(* CODESYS project PPC-GD-14.xml

Project tree, tasks and I/O mapping:
  Alarm Configuration
    alarm class Alarm (priority 30, acknowledge REP)
    alarm class Critical (priority 0, acknowledge ACK)
    alarm class Warning (priority 50, acknowledge REP)
    alarm group InverterComms
    alarm group Measurement
    alarm group Protection
    alarm group Startup
        0 []: Comparison Equal
    alarm group StopTrip
    alarm group SystemWatchdog
    AlarmStorage
    text list InverterComms
    text list Measurement
    text list Protection
    text list Startup
    text list StopTrip
    text list SystemWatchdog
  DataTypes/
    data type E_EventCode
    data type E_FailState
    data type E_MachineState
    data type E_ModbusResult
    data type E_StartupStatus
    data type ST_Energia
    data type ST_EventEntry
    data type ST_Medidor
    data type ST_Rele
    data type TTraceEntry
    data type UN_Convert_Word_To_Real
    data type UN_Energia
    data type UN_Medidor
    data type UN_Real_to_Word_array
    data type UN_Rele
  Eventos/
    function block FB_EventLog [ST]: Clear, GetEvent, LogEvent
  FB Controle/
    function block FB_Controle [ST]
    function block FB_Diagnostico [ST]
    function block FB_DroopP [ST]
    function block FB_FFQ [ST]
    function block FB_FLimiter [ST]
    function block FB_PAlloc [ST]
    function block FB_PI [ST]
    function block FB_PIQ [ST]
    function block FB_PowerController [ST]
    function block FB_QAlloc [ST]
    function block FB_SafetyMargin [ST]
    function block FB_Scheduler [ST]
  FB Escrita/
    function block FB_WriteInv [ST]
  FB Leitura/
    function block FB_ReadMedidor [ST]
    function block FB_ValidaDadosMedidor [ST]
    function block FB_ValidaDadosRele [ST]
  Variaveis/
    global variables Global
    global variables GVL_Alarm
    global variables GVL_EventLog
    global variables GVL_Persis
  function block FB_Startup [ST]
  program MainProgram [ST]
  FB da IHM/
    function block FB_EventDisplay [ST]
    function FC_EpochToString [ST]
    function FC_EventCodeToString [ST]
    function FC_SeverityToString [ST]
    function FC_UIntToHex16Sharp [ST]
*)

// DataTypes/E_EventCode
{attribute 'qualified_only'}
{attribute 'strict'}
// ════════════════════════════════════════════════════════════════════
// E_EventCode — Código unificado de eventos do PPC-GD
// ════════════════════════════════════════════════════════════════════
//
// FAIXAS DE CÓDIGOS:
//   0x0000          = Sem evento
//   0x1xxx          = INFO     (informações operacionais)
//   0x2xxx          = WARNING  (desvios toleráveis, sem ação de potência)
//   0x4xxx          = ALARM    (falhas que requerem atenção ou degradam)
//   0x8xxx          = CRITICAL (ações de segurança: FAIL_SAFE ou STOP)
//
// SUB-FAIXAS (2º nibble = módulo):
//   x0xx = Sistema / Geral
//   x1xx = Startup (FB_Startup)
//   x2xx = Medição (FB_ReadMedidor, FB_ValidaDadosRele)
//   x3xx = Comunicação inversores (FB_WriteInv)
//   x4xx = Controle (FB_Controle, FB_PowerController, FB_PIQ)
//   x5xx = Scheduler / Agenda
//   x6xx = Máquina de Estados (MainProgram)
//   x7xx = Proteção normativa (timers 15s/30s, hard-limit)
//   x8xx = STOP / Trip
//   x9xx = Reservado para expansão
//   xAxx = Erros gerados pelo Driver Modbus do Codesys
//
// Observação: códigos legados (ex-16#C1/C2/E1/E2/E3/F1) são referenciados
// por comentário e mapeados semanticamente, sem manter o mesmo valor numérico,
// para preservar a coerência de severidade por faixa.
// ════════════════════════════════════════════════════════════════════
TYPE E_EventCode :
(
    EVT_NONE                        := 16#0000,

    // ══════════════════════════════════════════════════════════════
    // INFO (0x1xxx) — registro operacional, sem ação
    // ══════════════════════════════════════════════════════════════

    // ── Startup ──
    INFO_STARTUP_BEGIN              := 16#1100,  // Inicialização iniciada
    INFO_SERIAL_COM_OK              := 16#1101,  // COM1 e COM2 prontos
    INFO_RTC_OK                     := 16#1102,  // Relógio lido com sucesso
    INFO_INVERTER_COUNT             := 16#1103,  // Contagem de inversores concluída
    INFO_INSTALLED_POWER            := 16#1104,  // Potência instalada calculada
    INFO_K1_CONFIRMED               := 16#1105,  // K1_in confirmado (debounce)
    INFO_K2_CONFIRMED               := 16#1106,  // K2_in confirmado (debounce)
    INFO_STARTUP_DONE               := 16#1107,  // Startup completo → operação

    // ── Operação normal ──
    INFO_MEDIDOR_READ_OK            := 16#1200,  // Leitura do medidor OK
    INFO_MEDIDOR_DATA_VALID         := 16#1201,  // Dados validados e filtro aplicado
    INFO_MEAS_RECOVERING            := 16#1202,  // contador nErrors reduzindo (opcional)

    // ── Escrita inversores (0x13xx)
    INFO_WRITE_INV_OK               := 16#1300,  // Escrita em inversor OK

    // ── Scheduler (0x15xx)
    INFO_SPECIAL_DATE_ACTIVE        := 16#1500,  // Data especial ativa na agenda
    INFO_ZERO_GRID_MODE             := 16#1501,  // Modo Zero Grid ativo

    // ── Recuperação / Reset ──
    INFO_CYCLE_COMPLETE             := 16#1600,  // Ciclo READ→CONTROL→WRITE→IDLE OK
    INFO_FAIL_RECOVERY              := 16#1601,  // Recuperação automática do FAIL
    INFO_STATE_CHANGE               := 16#1610,  // Transição de MachineState

    // ── STOP/Reset (0x18xx)
    INFO_STOP_K2_OPEN_CONFIRMED     := 16#1800,  // K2 confirmado aberto no STOP
    INFO_STOP_RESET_APPROVED        := 16#1801,  // Reset manual aprovado
    INFO_STOP_RESET_WAITING         := 16#1802,  // Aguardando Pt estável para reset

    // ══════════════════════════════════════════════════════════════
    // WARNING (0x2xxx) — desvio tolerável, sem ação de potência
    // ══════════════════════════════════════════════════════════════

    // ── Startup ──
    WARN_TC_POWER_NOT_SET           := 16#2100,  // TC_Power_kW não configurado
    WARN_NO_INVERSORES_COM02        := 16#2101,  // COM2 sem inversores (pode ser intencional)

    // ── Medição ──
    WARN_MEAS_USING_LAST_VALID      := 16#2200,  // Usando última medição válida
    WARN_MEAS_CROSS_CHECK_PA        := 16#2201,  // Validação cruzada Pa inconsistente
    WARN_MEAS_CROSS_CHECK_PB        := 16#2202,  // Validação cruzada Pb inconsistente
    WARN_MEAS_CROSS_CHECK_PC        := 16#2203,  // Validação cruzada Pc inconsistente
    WARN_MEAS_CROSS_CHECK_PT_SUM    := 16#2204,  // Pt ≠ Pa+Pb+Pc
    WARN_MEAS_CROSS_CHECK_PF        := 16#2205,  // PFt inconsistente com P/S
    WARN_MEAS_ERROR_ISOLATED        := 16#2206,  // Erro de medição isolado (1-4 erros)

    // ── Comunicação inversores ──
    WARN_WRITE_INV_ERROR            := 16#2300,  // Erro escrita em inversor individual
    WARN_WRITE_INV_TIMEOUT          := 16#2301,  // Timeout escrita em inversor individual

    // ── Controle ──
    WARN_P_ALLOC_SATURATED          := 16#2400,  // P alocado < P comandado
    WARN_Q_LIMITED_BY_SMAX          := 16#2401,  // Q limitado por Smax dos inversores
    WARN_PF_BELOW_TARGET            := 16#2402,  // PF < 0.92 (mas não por limite de S)
    WARN_PF_NOT_ACHIEVABLE          := 16#2403,  // PF impossível (banco de capacitor)
    WARN_PI_P_SATURATED             := 16#2404,  // PI de P saturado
    WARN_PI_Q_SATURATED             := 16#2405,  // PI de Q saturado
    WARN_PHASE_LIMITED              := 16#2406,  // Potência limitada por fase

    // ── Ciclo ──
    WARN_SCAN_OVERRUN               := 16#2600,  // Ciclo excedeu tolerância (1x)

          // ── STOP/reset
    WARN_STOP_RESET_DENIED          := 16#2800,  // Reset manual negado

    // ══════════════════════════════════════════════════════════════
    // ALARM (0x4xxx) — falha que requer atenção, pode degradar
    // ══════════════════════════════════════════════════════════════

    // ── Medição — Range ──
    ALARM_MEAS_VOLTAGE_A_RANGE      := 16#4200,  // Tensão fase A fora de faixa
    ALARM_MEAS_VOLTAGE_B_RANGE      := 16#4201,  // Tens  o fase B fora de faixa
    ALARM_MEAS_VOLTAGE_C_RANGE      := 16#4202,  // Tensão fase C fora de faixa
    ALARM_MEAS_CURRENT_A_RANGE      := 16#4203,  // Corrente fase A fora de faixa
    ALARM_MEAS_CURRENT_B_RANGE      := 16#4204,  // Corrente fase B fora de faixa
    ALARM_MEAS_CURRENT_C_RANGE      := 16#4205,  // Corrente fase C fora de faixa
    ALARM_MEAS_PT_RANGE             := 16#4206,  // Potência total fora de faixa
    ALARM_MEAS_PA_RANGE             := 16#4207,  // Potência fase A fora de faixa
    ALARM_MEAS_PB_RANGE             := 16#4208,  // Potência fase B fora de faixa
    ALARM_MEAS_PC_RANGE             := 16#4209,  // Potência fase C fora de faixa
    ALARM_MEAS_QT_RANGE             := 16#420A,  // Reativa total fora de faixa
    ALARM_MEAS_QA_RANGE             := 16#420B,  // Reativa fase A fora de faixa
    ALARM_MEAS_QB_RANGE             := 16#420C,  // Reativa fase B fora de faixa
    ALARM_MEAS_QC_RANGE             := 16#420D,  // Reativa fase C fora de faixa
    ALARM_MEAS_PFT_RANGE            := 16#420E,  // PF total fora de faixa
    ALARM_MEAS_PFA_RANGE            := 16#420F,  // PF fase A fora de faixa
    ALARM_MEAS_PFB_RANGE            := 16#4210,  // PF fase B fora de faixa
    ALARM_MEAS_PFC_RANGE            := 16#4211,  // PF fase C fora de faixa
    ALARM_MEAS_FROZEN               := 16#4212,  // Medição congelada (Pt sem variação)

    // ── Comunicação medidor ──
    ALARM_MEDIDOR_MODBUS_ERROR      := 16#4220,  // Erro Modbus do medidor
    ALARM_MEDIDOR_TIMEOUT           := 16#4221,  // Timeout leitura medidor

    // ── Comunicação inversores ──
    ALARM_COM_CH1_DEGRADED          := 16#4300,  // Canal COM1 >50% falhas
    ALARM_COM_CH2_DEGRADED          := 16#4301,  // Canal COM2 >50% falhas
	
	// Erros gerados pelo Driver Modbus do Codesys
    ALARM_MB_ILLEGAL_FUNC         	:= 16#4A01,
    ALARM_MB_ILLEGAL_ADDR         	:= 16#4A02,
    ALARM_MB_ILLEGAL_VALUE        	:= 16#4A03,
    ALARM_MB_SLAVE_FAILURE        	:= 16#4A04,
    ALARM_MB_ACKNOWLEDGE          	:= 16#4A05,
    ALARM_MB_SLAVE_BUSY           	:= 16#4A06,
    ALARM_MB_MEMORY_PARITY        	:= 16#4A08,
    ALARM_MB_GW_PATH_UNAVAIL      	:= 16#4A0A,
    ALARM_MB_GW_DEVICE_FAIL       	:= 16#4A0B,
    ALARM_MB_RESPONSE_TIMEOUT     	:= 16#4AA1,
    ALARM_MB_RESPONSE_CRC         	:= 16#4AA2,
    ALARM_MB_WRONG_SLAVE          	:= 16#4AA3,
    ALARM_MB_WRONG_FC             	:= 16#4AA4,
    ALARM_MB_TCP_WARMOR           	:= 16#4AA5,
    ALARM_MB_INVALID_DATA         	:= 16#4AA6,
    ALARM_MB_INVALID_PROTOCOL     	:= 16#4AA7,
    ALARM_MB_INVALID_HEADER       	:= 16#4AA8,
    ALARM_MB_INVALID_PARAM        	:= 16#4AA9,
    ALARM_MB_UNDEFINED            	:= 16#4AFF,
	ALARM_MB_APP_ABORTED          	:= 16#4AB1,
    ALARM_MB_APP_TIMEOUT          	:= 16#4AB2,

    // ══════════════════════════════════════════════════════════════
    // CRITICAL (0x8xxx) — ação de segurança (FAIL_SAFE ou STOP)
    // ══════════════════════════════════════════════════════════════

    // ── Startup ──
    CRIT_SERIAL_INIT_FAILED         := 16#8100,  // COM1/COM2 não inicializou
    CRIT_RTC_FAILED                 := 16#8101,  // Falha leitura RTC
    CRIT_NO_INSTALLED_POWER         := 16#8102,  // Potência instalada = 0
    CRIT_K1_TIMEOUT                 := 16#8103,  // K1 não respondeu (timeout)

    // ── Medição ──
    CRIT_MEAS_PERSISTENT_FAIL       := 16#8200,  // ex-16#C1 Medição com falha persistente (≥5 erros)
    CRIT_MEDIDOR_COM_FAIL           := 16#8201,  // ex-16#C2 Erro/Timeout Modbus medidor → FAIL

    // ── Comunicação inversores ──
    CRIT_COM_CHANNEL_FAIL           := 16#8300,  // ex-16#C2 Canal COM com falha total → FAIL

    // ── Controle ──
    CRIT_INSTALLED_POWER_ZERO       := 16#8400,  // InstalledPower = 0 em runtime → STOP

    // ── Scheduller ──
    CRIT_RTC_READ_FAIL              := 16#8500,  // RTC falhou durante operação
    CRIT_SCHEDULE_INDEX_INVALID     := 16#8501,  // Índice dia/hora inválido

    // ── Watchdog ──
    CRIT_SCAN_WATCHDOG              := 16#8600,  // ex-16#F1 3× overruns consecutivos → FAIL

    // ── Proteção normativa ──
    CRIT_HARD_LIMIT_15S             := 16#8700,  // ex-16#E1 P > LPI+10%Pnom por >15s → STOP
    CRIT_EXPORT_OVER_LPI_30S        := 16#8701,  // ex-16#E2 P > LPI por >30s → STOP
    CRIT_MEDIDOR_TIMEOUT_IN_FAIL    := 16#8702,  // ex-16#E3 30s sem medição válida em FAIL → STOP

    // ── STOP / Trip ──
    CRIT_STOP_ENTRY                 := 16#8800,  // Entrada no estado STOP
    CRIT_K2_DID_NOT_OPEN            := 16#8801,  // K2 não abriu após 2s → FaultLatch
    CRIT_STATE_CORRUPTION           := 16#8802   // MachineState inválido

) UINT;
END_TYPE

// DataTypes/E_FailState
{attribute 'qualified_only'}
{attribute 'strict'}
TYPE E_FailState :
(
    FS_INIT         := 0,  // Inicialização FAIL_SAFE
    FS_FORCE_ZERO   := 1,  // Forçar setpoint zero
    FS_WAIT_CONFIRM := 2,  // Aguardar confirmação escrita
    FS_VALIDATE     := 3,  // Validar geração zero
    FS_ESCALATE     := 4   // Escalar para STOP
) UINT;
END_TYPE

// DataTypes/E_MachineState
{attribute 'qualified_only'}
{attribute 'strict'}
TYPE E_MachineState :
(
	START       := 0,  // inicializa o sistema uma única vez
    IDLE        := 1,  // Aguardando condições de início
    READ        := 2,  // Lendo medidor
    CONTROL     := 3,  // Calculando setpoints
    WRITE       := 4,  // Enviando comandos inversores
    FAIL	    := 5,  // Redução forçada (sem trip)
    STOP        := 6,   // Trip + latch (reset manual)
	ERROR       := 255 // Estado inválido/corrupto (fallback)
) UINT;
END_TYPE

// DataTypes/E_ModbusResult
{attribute 'strict'}
TYPE E_ModbusResult :
(
    BUSY,   	// operação em andamento
    DONE,   	// leitura finalizada com sucesso (pulso curto)
    ERRO,   	// falha (permanece até reset)
	ABORT,		// comunicação foi abortada
	TIMEOUT,	// ocorreu TIMEOUT
	END			// finaliza a comunicação
);
END_TYPE

// DataTypes/E_StartupStatus
{attribute 'qualified_only'}
{attribute 'strict'}
TYPE E_StartupStatus :
(
  stSeriais,		(* inicializa serias COM1 e COM2 *)
  stInit,			(* inicializa variaveis *)
  stWait_K1,      	(* transição imediata quando o delay completa *)
  stWait_K2,       	(* mantém bK3_out; monitora bK2_in com debounce *)
  stDone,           (* sucesso: desliga bK3_out e liga bK4_out *)
  stError           (* erro: sinaliza e coloca saídas em estado seguro *)
);
END_TYPE

// DataTypes/ST_Energia
TYPE ST_Energia :
	STRUCT
		// variavel       tipo      modbusAddress origem         fator_escala 
		EAImp  : REAL := 0.0; // 101EH - energia ativa total positiva (kWh)
		Vazia1 : REAL := 0.0; // 1020H - void
		Vazia2 : REAL := 0.0; // 1022H - void
		Vazia3 : REAL := 0.0; // 1024H - void
		Vazia4 : REAL := 0.0; // 1026H - void
		EAExp  : REAL := 0.0; // 1028H - energia ativa total negativa (kWh)	
	END_STRUCT
END_TYPE

// DataTypes/ST_EventEntry
// ════════════════════════════════════════════════════════════════════
// ST_Event — Registro individual de evento no ring buffer
// ════════════════════════════════════════════════════════════════════
// Tamanho estimado: 28 bytes (verificar alinhamento no target)
//
// CAMPOS:
//   tTimestamp  — Epoch UTC (UDINT, até 2106). Obtido via SysTimeRtcGet.
//   eCode      — Código do evento (E_EventCode). Identifica unicamente o que ocorreu.
//   bRaised    — TRUE = evento apareceu / FALSE = evento foi limpo.
//                Permite rastrear par raise/clear no histórico.
//   rParam1    — Valor de contexto #1 no momento do evento.
//                Ex: Pt medido (kW) quando hard-limit disparou.
//   rParam2    — Valor de contexto #2 no momento do evento.
//                Ex: limite violado (kW), ou índice do inversor.
//   uMachState — Estado da máquina (E_MachineState) no momento do registro.
//                Essencial para análise pós-mortem.
// ════════════════════════════════════════════════════════════════════
TYPE ST_EventEntry :
STRUCT
    tTimestamp      : UDINT;            // UTC epoch (segundos)
    eCode           : E_EventCode;      // UINT — código unificado do evento
    bRaised         : BOOL;             // TRUE=raise, FALSE=clear
    rParam1         : REAL;             // contexto numérico #1
    rParam2         : REAL;             // contexto numérico #2
    uMachState      : UINT;             // E_MachineState no instante do registro
END_STRUCT
END_TYPE

// DataTypes/ST_Medidor
TYPE ST_Medidor :
	STRUCT
		//  22 variaveis do tipo real - ocupam 44 Words no array
		// variavel       tipo      modbusAddress origem         fator_escala 
		Ua    	    : REAL := 0.0; // 2006H - Tensão de fase A x 0,1 V
		Ub    	    : REAL := 0.0; // 2008H - Tensão de fase B x 0,1 V
		Uc    	    : REAL := 0.0; // 200AH - Tensão de fase C x 0,1 V
		Ia    	    : REAL := 0.0; // 200CH - Corrente de fase A x 0,001 A 
		Ib    	    : REAL := 0.0; // 200EH - Corrente de fase B x 0,001 A
		Ic    	    : REAL := 0.0; // 2010H - Corrente de fase C x 0,001 A
		Pt    	    : REAL := 0.0; // 2012H - Potencia ativa combinada x 0,1 W
		Pa    	    : REAL := 0.0; // 2014H - Potencia ativa fase A x 0,1 W
		Pb    	    : REAL := 0.0; // 2016H - Potencia ativa fase B x 0,1 W
		Pc    	    : REAL := 0.0; // 2018H - Potencia ativa fase C x 0,1 W	
		Qt    	    : REAL := 0.0; // 201AH - Potencia reativa combinada x 0,1 var
		Qa    	    : REAL := 0.0; // 201CH - Potencia reativa fase A x 0,1 var
		Qb    	    : REAL := 0.0; // 201EH - Potencia reativa fase B x 0,1 var
		Qc    	    : REAL := 0.0; // 2020H - Potencia reativa fase C x 0,1 var
		Reserved01  : REAL;        // 2022H - sem informação
		Reserved02  : REAL;        // 2024H - sem informação
		Reserved03  : REAL;        // 2026H - sem informação
		Reserved04  : REAL;        // 2028H - sem informação
		PFt    	    : REAL := 0.0; // 202AH - Fator de potência combinado (número positivo: indutivo, número negativo: capacitivo) (x  0,001)
		PFa    	    : REAL := 0.0; // 202CH - Fator de potência de fase A (número positivo: indutivo, número negativo: capacitivo)  (×0,001)
		PFb    	    : REAL := 0.0; // 202EH - Fator de potência de fase B (número positivo: indutivo, número negativo: capacitivo)  (×0,001)
		PFc    	    : REAL := 0.0; // 2030H - Fator de potência de fase C (número positivo: indutivo, número negativo: capacitivo)  (×0,001)
	END_STRUCT
END_TYPE

// DataTypes/ST_Rele
TYPE ST_Rele :
	STRUCT
		//  22 variaveis do tipo real - ocupam 44 Words no array
		// variavel       tipo      modbusAddress origem         fator_escala 
		Ua    	    : REAL := 0.0; // 2006H - Tensão de fase A x 0,1 V
		Ub    	    : REAL := 0.0; // 2008H - Tensão de fase B x 0,1 V
		Uc    	    : REAL := 0.0; // 200AH - Tensão de fase C x 0,1 V
		Ia    	    : REAL := 0.0; // 200CH - Corrente de fase A x 0,001 A 
		Ib    	    : REAL := 0.0; // 200EH - Corrente de fase B x 0,001 A
		Ic    	    : REAL := 0.0; // 2010H - Corrente de fase C x 0,001 A
		Pt    	    : REAL := 0.0; // 2012H - Potencia ativa combinada x 0,1 W
		Pa    	    : REAL := 0.0; // 2014H - Potencia ativa fase A x 0,1 W
		Pb    	    : REAL := 0.0; // 2016H - Potencia ativa fase B x 0,1 W
		Pc    	    : REAL := 0.0; // 2018H - Potencia ativa fase C x 0,1 W	
		Qt    	    : REAL := 0.0; // 201AH - Potencia reativa combinada x 0,1 var
		Qa    	    : REAL := 0.0; // 201CH - Potencia reativa fase A x 0,1 var
		Qb    	    : REAL := 0.0; // 201EH - Potencia reativa fase B x 0,1 var
		Qc    	    : REAL := 0.0; // 2020H - Potencia reativa fase C x 0,1 var
		Reserved01  : REAL;        // 2022H - sem informação
		Reserved02  : REAL;        // 2024H - sem informação
		Reserved03  : REAL;        // 2026H - sem informação
		Reserved04  : REAL;        // 2028H - sem informação
		PFt    	    : REAL := 0.0; // 202AH - Fator de potência combinado (número positivo: indutivo, número negativo: capacitivo) (x  0,001)
		PFa    	    : REAL := 0.0; // 202CH - Fator de potência de fase A (número positivo: indutivo, número negativo: capacitivo)  (×0,001)
		PFb    	    : REAL := 0.0; // 202EH - Fator de potência de fase B (número positivo: indutivo, número negativo: capacitivo)  (×0,001)
		PFc    	    : REAL := 0.0; // 2030H - Fator de potência de fase C (número positivo: indutivo, número negativo: capacitivo)  (×0,001)
	END_STRUCT
END_TYPE

// DataTypes/TTraceEntry
TYPE TTraceEntry :
STRUCT
        cyc         : UDINT;
        mode        : USINT;
        startEdge   : BOOL;
        xExecute    : BOOL;
        xAbort      : BOOL;
        xBusy       : BOOL;
        xDone       : BOOL;
        xError      : BOOL;
        xAborted    : BOOL;
        toQ         : BOOL;
        modbusErr   : UDINT;
        eResult     : E_ModbusResult;
    END_STRUCT
END_TYPE

// DataTypes/UN_Convert_Word_To_Real
TYPE UN_Convert_Word_To_Real :
	UNION
        Tw : ARRAY[0..1] OF WORD;
        Tr : REAL;
    END_UNION
END_TYPE

// DataTypes/UN_Energia
TYPE UN_Energia :
	UNION
        WordArray : ARRAY[0..11] OF WORD;
        EmReal    : ST_Energia;
    END_UNION
END_TYPE

// DataTypes/UN_Medidor
TYPE UN_Medidor :
	UNION
        WordArray : ARRAY[0..43] OF WORD;
        EmReal    : ST_Rele;
    END_UNION
END_TYPE

// DataTypes/UN_Real_to_Word_array
TYPE UN_Real_to_Word_array :
UNION
	RealArr  : ARRAY[1..15] OF REAL;   // 60 bytes
    WordArr  : ARRAY[1..30] OF WORD;   // 60 bytes
END_UNION
END_TYPE

// DataTypes/UN_Rele
TYPE UN_Rele :
	UNION
        WordArray : ARRAY[0..43] OF WORD;
        EmReal    : ST_Rele;
    END_UNION
END_TYPE

// Variaveis/Global
{attribute 'qualified_only'}
VAR_GLOBAL CONSTANT

    // Parâmetros do sistema
    SOFTVERSION          		: UINT := 21;   				// Versão da aplicação
	DATAAPLICATION				: DATE := DATE#2025-12-05;		// Data da aplicação
	NMAXINVERSORES				: UINT := 30;					// Capacidade máxima de inversores
	TIPOSINVERSORES				: UINT := 8;					// total de inversores diferentes que podem estar presentes
	NDATASESPECIAIS 			: UINT := 48; 					// Quantidade de datas especiais disponíveis ao todo (para 10 anos)
	TIMEZONEOFFSET				: DINT := -3; 			
    CYCLE_TIME_MS				: UDINT := 1000;  				// tempo de ciclo de controle
	CYCLE_TIME_TOLERANCE		: UDINT := 1100;  				// tolerancia de ultrapassagem para tempo de ciclo de controle de 10%

END_VAR

VAR_GLOBAL
	timestampUTC				: UDINT;
	Result 						: RTS_IEC_RESULT;
  	ControlCycle    			: REAL;            					// Tempo de ciclo de controle em SEGUNDOS (ex: 1.0 = 1 segundo)
	
	// Saidas digitais
  	K1_out  					: BOOL;   							// DI X5_1 - K1 - controle permissivo
	K2_out						: BOOL;								// DI X5_2 - K2 - controle trip
  	K3RedOut					: BOOL;								// DI X5_3 - nada pronto - acende vermelho
  	K4YellowOut  				: BOOL;   							// DI X5_4 - K2 aberto - acende amarelo
  	K5GreenOut  				: BOOL;   							// DI X5_5 - K2 fechou - acende verde
	K7OkOut  					: BOOL;   							// DI X5_7 - sinaliza ok
	K8ErroOut  					: BOOL;   							// DI X5_8 - sinaliza erro
		
	// Entredas digitais
	K1_in        				: BOOL;                				// DI X12_1 - contato auxliar de K1
  	K2_in        				: BOOL;                				// DI X12_2 - contato auxliar de K2

    //    Medições (REAL) - Tensões (V), Correntes (A), Potências Ativas (W), Potências Reativas (var), PF (adimensional, sinal: + indutivo, - capacitivo)
	
    Ua  			: REAL := 0.0; // Tensão de fase A   - 2006H - Tensão de fase A em Volts (x 0,1 V)
    Ub  			: REAL := 0.0; // Tensão de fase B   - 2008H - Tensão de fase B em Volts (x 0,1 V)
    Uc  			: REAL := 0.0; // Tensão de fase C   - 200AH - Tensão de fase C em Volts (x 0,1 V)
	
	Ia    			: REAL 	:= 0.0; // 200CH - Corrente de fase A em A (x 0,001 A) 
	Ib    			: REAL 	:= 0.0; // 200EH - Corrente de fase B em A (x 0,001 A) 
	Ic    			: REAL 	:= 0.0; // 2010H - Corrente de fase C em A (x 0,001 A) 
	
	Pt    			: REAL 	:= 0.0; // 2012H - Potencia ativa combinada em kW (x 0.1 para W, x 0.0001 para kW)
	Pa    			: REAL 	:= 0.0; // 2014H - Potencia ativa fase A 	em kW (x 0.1 para W, x 0.0001 para kW)
	Pb    			: REAL 	:= 0.0; // 2016H - Potencia ativa fase B 	em kW (x 0.1 para W, x 0.0001 para kW)
	Pc    			: REAL 	:= 0.0; // 2018H - Potencia ativa fase C    em kW (x 0.1 para W, x 0.0001 para kW)

	Qt    			: REAL 	:= 0.0; // 201AH - Potencia reativa combinada em kvar (x 0.1 para var, x 0.0001 para kvar)
	Qa    			: REAL 	:= 0.0; // 201CH - Potencia reativa fase A	 em kvar (x 0.1 para var, x 0.0001 para kvar)
	Qb    			: REAL 	:= 0.0; // 201EH - Potencia reativa fase B	 em kvar (x 0.1 para var, x 0.0001 para kvar)
	Qc    			: REAL 	:= 0.0; // 2020H - Potencia reativa fase C	 em kvar (x 0.1 para var, x 0.0001 para kvar)
	
	PFt    			: REAL 	:= 0.0; // 202AH - Fator de potência combinado (número positivo: indutivo, número negativo: capacitivo) (x0,001)
	PFa    			: REAL 	:= 0.0; // 202CH - Fator de potência de fase A (número positivo: indutivo, número negativo: capacitivo) (x0,001)
	PFb    			: REAL 	:= 0.0; // 202EH - Fator de potência de fase B (número positivo: indutivo, número negativo: capacitivo) (x0,001)
	PFc    			: REAL 	:= 0.0; // 2030H - Fator de potência de fase C (número positivo: indutivo, número negativo: capacitivo) (x0,001)	

    //   COMANDOS E TELEMETRIA - Saídas do Controle 
	
	// definição dos inversores dos dois canais de comunicação
	
	trigInvCOM100  	: ARRAY[1..15] OF BOOL;
    pInversores100 	: ARRAY [1..15] OF POINTER TO ModbusSlaveComPort; 				// array de pointers para Inversor01..Inversor15 (apenas ponteiros - não recria instâncias)
	trigMedidor100 	: BOOL;
	pMedidor100		: POINTER TO ModbusSlaveComPort;
	
	trigInvCOM200  	: ARRAY[1..15] OF BOOL;
	pInversores200 	: ARRAY [1..15] OF POINTER TO ModbusSlaveComPort; 				// array de pointers para Inversor01..Inversor15 (apenas ponteiros - não recria instâncias)
	trigMedidor200 	: BOOL;
	pMedidor200		: POINTER TO ModbusSlaveComPort;
	
	// Potencia Total instalada e potencia Aparente Total instalada
  	InstalledPower 	: REAL; 														// Soma da potência nominal de todos os inversores ativos
	Q_max_permitido : REAL := 0.0;    												// Q máximo permitido (kvar)
	InstalledSmax   : REAL; 														// NOVO: Potência Aparente Máxima Total (kVA)	
	
	// COMANDOS DE CONTROLE
	MaxExportLimit 	: REAL;              											// Limite de exportação do scheduler (kW)
	P_cmd_total_kW 	: REAL;              											// Comando total de P (kW)
	Q_cmd_total_kvar: REAL;            												// Comando total de Q (kvar)
	
    
    // Telemetria: Setpoint atual da agenda (antes das proteções)
    TotalPowerPercent : REAL;

    // Telemetria: Potência Reativa total desejada (kVA)
    TotalReactivePower : REAL;

    // Telemetria: Valores efetivos calculados para cada inversor
    P_inv_kW     	: ARRAY[1..NMAXINVERSORES] OF REAL; 							// valor de setpoint de potencia ativa em kW
	P_inv_Percent 	: ARRAY[1..NMAXINVERSORES] OF REAL; 							// valor de setpoint de potencia ativa em percentual do nominal
    Q_inv_kvar    	: ARRAY[1..NMAXINVERSORES] OF REAL; 							// valor de setpoint de potencia reativa em kVA
    PF_inv 			: ARRAY[1..NMAXINVERSORES] OF REAL; 							// valor do fator de potencia de cada inversor (deve ser 0,92 para todos)
	P_inv_limit 	: ARRAY[1..NMAXINVERSORES] OF REAL; 							// valor limite de potencia ativa com base na SMAX de cada um
	
	// Margem de segurança para compensar erro de TC perto de zero, o sistema tentará manter importação mínima garantido que não haja exportação
	SafetyMargin_pct: REAL :=0.03;
	TC_Power_kW		: REAL := 0.0; // deve ser configurado como 3% da potencia total sob controle pelo TC
	
	// ════════════════════════════════════════════════════════════════
	// DIAGNÓSTICO DE PF
	// ════════════════════════════════════════════════════════════════
	Q_available_max : REAL;             											// Q máximo disponível (kvar)
	PF_effective 	: REAL;                											// PF efetivo resultante
	PFErro 			: BOOL;                   										// TRUE = PF < 0.92 não atingível (banco de capacitores)
    
	// ════════════════════════════════════════════════════════════════
    // DIAGNÓSTICO DE FATOR DE POTÊNCIA
    // ════════════════════════════════════════════════════════════════
    
    // Status geral
    PF_target : REAL := 0.92;                   // PF alvo (mínimo aceitável)
    PF_measured : REAL;                         // PF medido no ponto de conexão
    PF_achieved : REAL;                         // PF efetivamente alcançado após compensação
    PF_OK : BOOL;                               // TRUE = PF ≥ 0.92
    
    // Potências
    P_generated_kW : REAL;                      // P total gerado pelos inversores
    P_allocated_kW : REAL;                      // P efetivamente alocado
    Q_measured_kvar : REAL;                     // Q medido no ponto de conexão (carga)
    Q_required_kvar : REAL;                     // Q necessário para atingir PF ≥ 0.92
    Q_commanded_kvar : REAL;                    // Q comandado pelo FB_PIQ
    Q_available_kvar : REAL;                    // Q que inversores conseguem fornecer
    Q_allocated_kvar : REAL;                    // Q efetivamente alocado
    Q_deficit_kvar : REAL;                      // Déficit de Q (se > 0, falta Q)
    
    // Capacidade dos inversores
    S_total_available_kVA : REAL;               // S total disponível (soma de todos inversores)
    S_total_used_kVA : REAL;                    // S total utilizado
    S_utilization_pct : REAL;                   // % de utilização de S
    Q_capacity_total_kvar : REAL;               // Capacidade total de Q dos inversores (atual)
    Q_utilization_pct : REAL;                   // % de utilização de Q
    
    // Diagnóstico e recomendações
    Q_deficit_percent : REAL;                   // Déficit de Q em % do necessário
    Capacitor_bank_size_kvar : REAL;            // Tamanho recomendado de banco de capacitores
    Capacitor_bank_recommended : BOOL;          // TRUE = Recomenda banco de capacitores
    PF_alarm_code : UINT;                       // Código de alarme (0=OK, 1=Aviso, 2=Crítico)
    PF_alarm_message : STRING(255);             // Mensagem descritiva do alarme
    
    // Histórico (opcional)
    PF_min_24h : REAL := 1.0;                   // PF mínimo nas últimas 24h
    PF_avg_24h : REAL := 1.0;                   // PF médio nas últimas 24h
    Q_deficit_max_24h : REAL;                   // Déficit máximo de Q nas últimas 24h
    PF_alarm_count_24h : UDINT;                 // Quantidade de alarmes nas últimas 24h
    
    // Inversores individuais (diagnóstico detalhado)
    Inv_S_utilization : ARRAY[1..NMAXINVERSORES] OF REAL;  // % S usado por inversor
    Inv_Q_available : ARRAY[1..NMAXINVERSORES] OF REAL;    // Q disponível por inversor (kvar)
    Inv_limited : ARRAY[1..NMAXINVERSORES] OF BOOL;        // TRUE = Inversor limitado por S	
END_VAR

// Variaveis/GVL_Alarm
{attribute 'qualified_only'}
VAR_GLOBAL
    // ─────────────────────────────────────────────────────────
    // ALARM MANAGER FLAGS (condições booleanas)
    // ─────────────────────────────────────────────────────────
    // Medição / Medidor
    ALM_MEAS_MEDIDOR_TIMEOUT       	: BOOL := FALSE;  // timeout de leitura (READ)
    ALM_MEDIDOR_MODBUS_ERRO        	: BOOL := FALSE;  // xError do medidor (READ)
    ALM_MEAS_PERSISTENT_FAIL		: BOOL := FALSE;  // bPoucosErros = FALSE
    ALM_MEAS_FROZEN	                : BOOL := FALSE;  // diagnosticCode = A900 (se aplicável)
    ALM_MEAS_USING_LAST_VALUEU		: BOOL := FALSE;  // bPoucosErros=TRUE e bDadosOK=FALSE
	ALM_MEAS_RANGE_ERROR    		: BOOL := FALSE;    // Warning: Valor fora de faixa
    ALM_MEAS_XCHECK_FAIL   			: BOOL := FALSE;    // Warning: Validação cruzada falhou

    // Comunicação inversores
    ALM_MODBUS_COM1_FAIL        	: BOOL := FALSE;  // >50% falhas COM1 no ciclo
    ALM_MODBUS_COM2_FAIL            : BOOL := FALSE;  // >50% falhas COM2 no ciclo
    ALM_COM_CHANNEL_FAIL           	: BOOL := FALSE;  // falha geral de comunicação → FAIL/STOP

    // Sistema
	ALM_SCAN_OVERRUN        		: BOOL := FALSE;    // Warning: Watchdog de ciclo
    ALM_RTC_FAIL            		: BOOL := FALSE;    // Error: Falha RTC
    ALM_NO_INVERTERS        		: BOOL := FALSE;    // Error: Nenhum inversor configurado
    ALM_INSTALLED_PWR_ZERO  		: BOOL := FALSE;    // Error: Potência instalada = 0
    ALM_TC_POWER_NOT_SET            : BOOL := FALSE;    // PerVar.TC_Power_kW = 0 na inicialização

    // Proteções normativas
    ALM_HARDLIMIT_15S       		: BOOL := FALSE;    // Error: P > LPI+10% por >15s
    ALM_EXPORT_30S          		: BOOL := FALSE;    // Error: P > LPI por >30s
    ALM_K2_NOT_OPENED       		: BOOL := FALSE;    // Error: K2 não abriu após trip
	
	// Status do sistema
    ALM_STOP_ACTIVE	                : BOOL := FALSE;  	// MachineState=STOP
	ALM_FAIL_ACTIVE					: BOOL := FALSE;  	// MachineState=FAIL

    // ── Controle / PF ──
    ALM_PF_BELOW_TARGET     		: BOOL := FALSE;    // Warning: PF < 0.92
    ALM_PF_CRITICAL         		: BOOL := FALSE;    // Error: PF < 0.92 + Q saturado
    ALM_Q_SATURATED         		: BOOL := FALSE;    // Info: Q limitado por S
END_VAR

// Variaveis/GVL_EventLog
{attribute 'qualified_only'}
// ════════════════════════════════════════════════════════════════════
// GVL_EventLog — Constantes do sistema de log de eventos
// ════════════════════════════════════════════════════════════════════
// Autor: Eng. Principal / Revisão Técnica PPC-GD
// Plataforma: WAGO CC100 (751-9402) / CODESYS V3.5 SP21 Patch 4
//
// DIMENSIONAMENTO:
//   64 entradas × 28 bytes = ~1.792 bytes de RETAIN
//   WAGO CC100 possui ~32 kB RETAIN → uso < 6%
//   Com ~1 evento/min, cobre >1 hora de histórico completo
//   Com taxa de pico (~10 eventos em cascata), ainda retém >6 min
// ════════════════════════════════════════════════════════════════════
{attribute 'qualified_only'}
VAR_GLOBAL CONSTANT
    MAX_EVENT_ENTRIES   : UINT := 64;   // Tamanho do ring buffer (potência de 2 facilita debug)
END_VAR

// Variaveis/GVL_Persis
{attribute 'qualified_only'}
VAR_GLOBAL PERSISTENT RETAIN

    // CONFIGURAÇÕES DO SISTEMA (Dados que não podem ser perdidos no desligamento)
    
    // --- Configuração dos Inversores ---
	NInversoresCOM01    : UINT :=0;
	NInversoresCOM02    : UINT :=0;
	
    // Potência nominal (kW) por tipo
    InvActivePower 		: ARRAY[1..Global.NMAXINVERSORES] OF REAL; 		// kW
    // Potência Aparente Máxima (kVA) por tipo 
    InvSmaxPower 		: ARRAY[1..Global.NMAXINVERSORES] OF REAL;		// kVA

    // --- Parâmetros de Controle de Exportação ---
    PowerMode 			: UINT := 2;      								// 0=Total, 1=Por Fase, 2=Ambos
	OperationMode		: BOOL := TRUE;									// FALSE=Export Control  TRUE=Zero Grid
	ControlMode			: UINT := 1;									// 0 = manual  1 = automatico (PI ativo)
    TotalMaxExport_kW 	: REAL := 0; 									// Limite físico total (kW)
    PhaseMaxExport_kW 	: REAL := 0; 									// Limite físico por fase (kW)

    (* 
	Regra prática para GD solar: Ti entre 5s e 20s. Mais rápido pode oscilar com a latência Modbus. 
	Mais lento perde capacidade de compensar nuvens passando.
	Ti é o Tempo Integral do controlador PI, também chamado de tempo de reset.
	Relação Ki= Kp / Ti   Então se você tem Kp = 1.0 e Ti = 10s => Ki=1.0/10 = 0.1 (por segundo)
	Na prática para seu sistema:
	Ti pequeno (ex: 2s) → integral age rápido → mais agressivo → risco de oscilação
	Ti grande (ex: 30s) → integral age devagar → mais conservador → lento para corrigir erro estacionário
	Ti = 10s → o controlador elimina o erro estacionário em aproximadamente 30 a 40 segundos (≈ 3-4 × Ti)
	Resumo em uma frase:
	Ti = 10s é "quanto tempo o integrador leva para alcançar a mesma força que o proporcional já deu instantaneamente".
	*)
	
	// --- Controle Droop (Potência Ativa) ---
	Droop_Enable     	: BOOL := TRUE;      							// Habilita droop
	K_Droop          	: REAL := 0.15;      							// kW/kW  (ex.: 0.05 = 5% de ganho)
	Deadband_Droop   	: REAL := 2.0;       							// % (erro menor não gera droop)
	Droop_Max        	: REAL := 0.4;       							// Fração da potência instalada (ex.: 0.6 = 60%)
	
	// --- Parâmetros do Controlador PI (Potência Ativa) ---
    Kp_P           		: REAL := 0.25;									// Recomendado: 0.1 a 1.0
																	    // Maior → resposta mais rápida, risco de oscilação
																	    // Menor → mais suave, mas mais lento
    Ki_P           		: REAL := 0.02;									// Recomendado: 0.02 a 0.1 - Com 1s de ciclo e tempo morto ~1,2–1,6s, integral muito alto oscila.
																		// Com T=1s: constante de tempo integral Ti = Kp/Ki = 12,5s
																	    // Significado: elimina erro estacionário em ~10 segundos
																	    // NUNCA > 0.2 com T=1s (oscilação garantida)
	RampUp_P 			: REAL := 15.0;           						// Rampa de subida (kW/s) - limitar a 15-20 kW/s por causa do sweep de setpoints nos inversores
	RampDown_P 			: REAL := 20.0;         						// Rampa de descida (kW/s) - RampDown_P ≤ 20–30 kW/s
    Deadband_P  		: REAL := 1.0;  								// % da potência instalada (ex: 1.0 = 1%)
	
    // --- Configuração de Fator de Potência (PF) e Reativos (Q) ---
    PF_target       	: REAL := 0.92; 								// Alvo |PF|
	PF_sign				: REAL := 1.0;
    // Parâmetros do PI de Correção de Q (Feedforward + Feedback)
    Kp_Q           		: REAL := 50.0;									// Recomendado: 20.0 a 100.0 kvar/pu_PF
																	    // Unidade: kvar por unidade de erro de PF
																	    // Ex: erro PF = 0.02 → P_term = 50 * 0.02 = 1.0 kvar
    Ki_Q           		: REAL := 5.0;									// Recomendado: 2.0 a 10.0 kvar/(pu_PF·s
																	    // Com T=1s: Ti = Kp/Ki = 10s => elimina erro em ~30-40s
																	    // Significado: corrige PF em ~10 segundos	
	RampUp_Q 			: REAL := 50.0;            						// Rampa de subida (kvar/s)
	RampDown_Q 			: REAL := 50.0;          						// Rampa de descida (kvar/s)
	Deadband_Q 			: REAL := 0.01;          						// Zona morta de PF (ex: 0.01 = ±0.01) — padrão para GD

    // --- Histerese de Habilitação ---
    HysteresisOn	   	: REAL := 0.01; 								// Liga controle acima de 1%
    HysteresisOff		: REAL := 0.01; 								// Desliga abaixo de 1%
		
    // --- Agenda Semanal (7 dias x 24 horas) e Datas Especiais
	bHorarioVerao 		: BOOL:= FALSE;									// se TRUE  = Horário de Verão Ativo (+1h)
    WeekSchedule_kW 	: ARRAY[1..7, 1..24] OF REAL; 					// (1=Dom 2=Seg 3=Ter 4=Quarta 5=Quinta 6=Sexta 7=Sábado) em kW
    DatasEspeciais   	: ARRAY[1..GLOBAL.NDATASESPECIAIS] OF DATE;		// inicializa com zeros
	SpecialDaySchedule 	: ARRAY[1..Global.NDATASESPECIAIS] OF REAL;		// cada data especial tem apenas um valor de potencia maxima valido para o dia inteiro

    // ════════════════════════════════════════════════════════════════
    // LIMITES FÍSICOS DO SISTEMA (Baseados no Transformador e Rede)
    // ════════════════════════════════════════════════════════════════
	// SafetyMargin_kW = SafetyMargin_pct × TC_Power_kW / 100 - Margem de segurança para compensar erro de TC perto de zero
	SafetyMargin_pct 	: REAL := 3.0;     								// Percentual do TC (%)
	// Exemplo 1: TC de 500 A, Tensão 380 V => P_TC = √3 × V × I = 1.732 × 380 × 500 = 329 kW
	TC_Power_kW			: REAL := 0.0; 									// deve ser configurado como 3% da potencia total sob controle pelo TC
	
	VMIN 				: REAL := 7170;  // Volts - tensão de fase minima para tensão primária de 13,8kV
    VMAX 				: REAL := 8370;  // Volts - tensão de fase máxima para tensão primária de 13,8kV
    IMAX 				: REAL := 125.0;  // Amperes - corrente de linha - para potencia de usina de 3MW erro transformador 5%
    PMAX 				: REAL := 3200.0; // kW (Demanda contratada + 10% de margem)
	QMAX				: REAL := 2400.0; // kvar tan(acos(0.8)) × Pmax
	// τ = tempo para atingir ~63% do valor final e T_scan = período de amostragem (1s no seu caso)
	// α = T_scan / (τ + T_scan)  => Alpha=0.5 => 3 segundos para atingir 95% do valor final
	// Item 2.1: "Responder em até 15 segundos a rejeição de carga"
	// Item 2.2: "Limitar exportação em até 15 segundos"
	// Nuvens passageiras: variação em 1–5 segundos
	// Rejeição de carga: instantânea (< 1s)
	// Ruído de medição: < 100 ms
	ALPHA				: REAL := 0.25;
	
END_VAR

// FB_Startup
(* FB: fbStartup
   1) Ativa K1_out
   2) Aguarda 400 ms antes de verificar se K1_in está ativo
      -> Se K1_in NÃO estiver ativo depois deste tempo, sinaliza erro e sai da fbStartup
   3) Monitorar K2_in com debounce até ficar ativo 
   4) Enquanto aguarda K2_in ativar, mantém K4_out ativo
   5) Quando K2_in ativar (após debounced), desativa K4_out e ativa K5_out
   6) O controlador aguarda até K2_in = TRUE
   Notas:
   	- IMPORTANTE: se não forem usados contados auxiliares nos disjuntores, K1_in e K2_in precisam ser conectados a 24V
	- Este FB apenas sinaliza os outputs K1_out, K3_out, K4_out e K5_out.
   	- Implementado com máquina de estados e TONs (tDelay e tDebounce). TON deve ser chamado toda iteração.  *)
   
FUNCTION_BLOCK FB_Startup
VAR_OUTPUT
  stState			: E_StartupStatus:= E_StartupStatus.stSeriais;
END_VAR

VAR
  fbChannel       	: ModbusChannel;
  debouncedK1     	: BOOL := FALSE;   								// flag auxiliar informando que K1_in está estável em 1 
  TonDebounceK1     : TON;                          				// Novo timer debounce K1_in
  TimeDebounceK1    : TIME := T#500MS;              				// Tempo de debounce para K1

  debouncedK2 		: BOOL := FALSE; 								// flag auxiliar informando que K2_in está estável em 1 
  TonDebounceK2 	: TON;   										// timer para debounce de bk2 
  TimeDebounceK2    : TIME := T#500MS;     							// tempo de debounce para leitura de K2_in 
  
  cmdK01     		: BOOL := FALSE;  								// comandos calculados por ciclo e aplicados no final 
  auxRed     		: BOOL := FALSE;
  auxYellow     	: BOOL := FALSE;
  auxGreen     		: BOOL := FALSE;
  auxK1_in  		: BOOL;											// entradas digitais lidas no inicio da função 
  auxK2_in			: BOOL;
  indice			: UINT;
  
  // Variáveis para o Master 01 (COM1)
  eDeviceState01     		: DED.DEVICE_STATE; 					// Para guardar o estado retornado
  xDiagInfoIsAvailable01 	: BOOL;            						// Para guardar a saída xDiagnosisInfoAvailable
  eError01	      	    	: DED.ERROR;        					// Para guardar o código de erro
  xMaster01IsReady   		: BOOL;            						// Nosso booleano final de "pronto"
  
  // Variáveis para o Master 02 (COM2)
  eDeviceState02     		: DED.DEVICE_STATE; 					// Para guardar o estado retornado
  xDiagInfoIsAvailable02 	: BOOL;            						// Para guardar a saída xDiagnosisInfoAvailable
  eError02	           		: DED.ERROR;        					// Para guardar o código de erro
  xMaster02IsReady   		: BOOL;            						// Nosso booleano final de "pronto"
 

END_VAR

// INICIA AQUI

auxK1_in := Global.K1_in;
auxK2_in := Global.K2_in;

TonDebounceK1(IN := (stState = E_StartupStatus.stWait_K1) AND auxK1_in, PT := TimeDebounceK1); 	// debounce para K1_in
TonDebounceK2(IN := (stState = E_StartupStatus.stWait_K2) AND auxK2_in, PT := TimeDebounceK2);  // debounce para K2_in

CASE stState OF 																				// Máquina de estados

	E_StartupStatus.stSeriais:
		eDeviceState01 := Master_01.GetDeviceState(
			xDiagnosisInfoAvailable => xDiagInfoIsAvailable01,
			eError                  => eError01
			);
		eDeviceState02 := Master_02.GetDeviceState(
			xDiagnosisInfoAvailable => xDiagInfoIsAvailable02,
			eError                  => eError02
			);
  		xMaster01IsReady := (eDeviceState01 = DED.DEVICE_STATE.RUNNING); 
   		xMaster02IsReady := (eDeviceState02 = DED.DEVICE_STATE.RUNNING); 
		
		IF xMaster01IsReady AND xMaster02IsReady THEN
			stState := E_StartupStatus.stInit;
		ELSE
			stState := E_StartupStatus.stSeriais;
			// dispara Alarme por não conseguir abrir seriais
		END_IF
		
  	E_StartupStatus.stInit:																		// Inicialização única
	   
		cmdK01 			:= FALSE;
		auxRed  		:= FALSE;
		auxYellow 		:= FALSE;
		auxGreen  		:= FALSE;
		debouncedK1 	:= FALSE;
		debouncedK2 	:= FALSE;
		
		// Testa leitura do relógio do sistema na inicialização
		Global.timestampUTC := TO_UDINT(SysTimeRtcGet(Global.Result)); 							// UDINT#1528268918
		IF Global.Result <> eResultCode.OK THEN 												// Em caso de erro de leitura do relógio, zera a saída por segurança
			// sinalizar que houve erro para ler o relógio
			Global.K8ErroOut:=TRUE;
			RETURN;
		END_IF
	
		// Porta de comunicação COM1
		Global.pMedidor100   		:= ADR(Medidor100);
		Global.pInversores100[1]  	:= ADR(Inversor101);
		Global.pInversores100[2]  	:= ADR(Inversor102);
		Global.pInversores100[3]	:= ADR(Inversor103);
		Global.pInversores100[4] 	:= ADR(Inversor104);
		Global.pInversores100[5]	:= ADR(Inversor105);
		Global.pInversores100[6] 	:= ADR(Inversor106);
		Global.pInversores100[7] 	:= ADR(Inversor107);
		Global.pInversores100[8] 	:= ADR(Inversor108);
		Global.pInversores100[9] 	:= ADR(Inversor109);
		Global.pInversores100[10]	:= ADR(Inversor110);
		Global.pInversores100[11]	:= ADR(Inversor111);
		Global.pInversores100[12] 	:= ADR(Inversor112);
		Global.pInversores100[13] 	:= ADR(Inversor113);
		Global.pInversores100[14] 	:= ADR(Inversor114);
		Global.pInversores100[15] 	:= ADR(Inversor115);
		
		// Porta de comunicação COM2
		Global.pMedidor200   	  	:= ADR(Medidor200);
		Global.pInversores200[1]  	:= ADR(Inversor201);
		Global.pInversores200[2]  	:= ADR(Inversor202);
		Global.pInversores200[3]  	:= ADR(Inversor203);
		Global.pInversores200[4]  	:= ADR(Inversor204);
		Global.pInversores200[5] 	:= ADR(Inversor205);
		Global.pInversores200[6]  	:= ADR(Inversor206);
		Global.pInversores200[7]  	:= ADR(Inversor207);
		Global.pInversores200[8]  	:= ADR(Inversor208);
		Global.pInversores200[9]  	:= ADR(Inversor209);
		Global.pInversores200[10] 	:= ADR(Inversor210);
		Global.pInversores200[11] 	:= ADR(Inversor211);
		Global.pInversores200[12] 	:= ADR(Inversor212);
		Global.pInversores200[13] 	:= ADR(Inversor213);
		Global.pInversores200[14] 	:= ADR(Inversor214);
		Global.pInversores200[15] 	:= ADR(Inversor215);
		
		FOR indice := 1 TO 15 DO														// inicialização dos canais de comunicação
			fbChannel(Slave := Global.pInversores100[indice]^,xExecute := FALSE,xAbort := FALSE,iChannelIndex := 0);
			fbChannel(Slave := Global.pInversores200[indice]^,xExecute := FALSE,xAbort := FALSE,iChannelIndex := 0); 
		END_FOR
	
		// =========================================================================================
		// 0. PREPARAÇÃO DO TEMPO DE CICLO - feito na inicialização
		// =========================================================================================
		// Converte TIME (ex: T#500ms) para REAL (0.5 segundos) para uso nos PIDs
		Global.ControlCycle := UDINT_TO_REAL(Global.CYCLE_TIME_MS)/1000;  				// converte para segundos
			
		// ============================================================
		// CONTAGEM AUTOMÁTICA DE INVERSORES (sequencial por potência)
		// ============================================================
		
		// COM1: índices 1..15
		GVL_Persis.NInversoresCOM01 := 0;
		FOR indice := 1 TO 15 DO
			IF GVL_Persis.InvActivePower[indice] > 0.0 THEN
				GVL_Persis.NInversoresCOM01 := indice;   // mantém maior índice válido
			ELSE
				EXIT;  // encontrou buraco -> encerra contagem
			END_IF
		END_FOR
		
		// COM2: índices 16..30
		GVL_Persis.NInversoresCOM02 := 0;
		FOR indice := 16 TO 30 DO
			IF GVL_Persis.InvActivePower[indice] > 0.0 THEN
				GVL_Persis.NInversoresCOM02 := indice - 15;   // converte para faixa 1..15
			ELSE
				EXIT;  // encontrou buraco -> encerra contagem
			END_IF
		END_FOR		
		
		// =========================================================================================
		// 1. CÁLCULO DA POTÊNCIA INSTALADA TOTAL (Ativa e Aparente)  - feito na inicialização
		// =========================================================================================
		// Soma a capacidade nominal de todos os inversores configurados.
		// Isso permite mudar a planta dinamicamente sem recompilar.
		
		Global.InstalledPower := 0.0;
		Global.InstalledSmax  := 0.0;
		
		FOR indice := 1 TO Global.NMAXINVERSORES DO
			// Soma Potência Ativa Máxima (kW)
			Global.InstalledPower := Global.InstalledPower + GVL_Persis.InvActivePower[indice];
			// Soma Potência Aparente Máxima (kVA)
			Global.InstalledSmax := Global.InstalledSmax + GVL_Persis.InvSmaxPower[indice];
		END_FOR

		// Se não houver inversores ou potência válida, zera tudo e sai.
		IF Global.InstalledPower <= 0.0 THEN
			Global.TotalReactivePower := 0.0;
			// SINALIZA ALARME
			Global.K8ErroOut:=TRUE;
			RETURN;
		END_IF
		
		// Calcula Q_max_permitido 
	    Global.Q_max_permitido := Global.InstalledPower * 0.4256;  // tan(acos(0.92))
			
		// Configura TC_Power_kW se não foi configurado
		IF GVL_Persis.TC_Power_kW = 0.0 THEN
			// SINALIZA ALARME
			Global.K8ErroOut:=TRUE;
			GVL_Persis.TC_Power_kW := Global.InstalledPower;  // Aproximação conservadora
		END_IF

		// Muda para próximo estado	
		stState := E_StartupStatus.stWait_K1;

  E_StartupStatus.stWait_K1:															// DEBOUNCE K1
  
		cmdK01 := TRUE;
		auxRed := TRUE;																	// Status: aguardando K1 com debounce
		auxYellow := FALSE;
		auxGreen := FALSE;
		IF TonDebounceK1.Q THEN
		  debouncedK1 := TRUE;
		ELSE
		  debouncedK1 := FALSE;
		END_IF
	
		IF debouncedK1 THEN
		  stState := E_StartupStatus.stWait_K2;												// Somente avança se K1 está estabilizado
		  debouncedK2 := FALSE;
		  TonDebounceK1(IN := FALSE, PT := TimeDebounceK1); 								// (Opcional) reseta timer
		  auxRed := FALSE;																	// Status: aguardando K1 com debounce
		  auxYellow := TRUE;
		  auxGreen := FALSE;
		  
		END_IF

  E_StartupStatus.stWait_K2:	
  
		IF TonDebounceK2.Q THEN																// tDebounce.Q será TRUE se K2_in estável
		  debouncedK2 := TRUE;
		ELSE     																					
		  debouncedK2 := FALSE;																// se K2_in voltar a false, reseta timer
		END_IF
	
		IF debouncedK2 THEN
		  stState := E_StartupStatus.stDone;												// K2_ok e estável, processo de startup completo
		  TonDebounceK2(IN := FALSE, PT := TimeDebounceK2); 								// (Opcional) reseta timer
		  auxRed := FALSE;																	// Status: aguardando K1 com debounce
		  auxYellow := FALSE;
		  auxGreen := TRUE;
		END_IF
	
	E_StartupStatus.stDone:
	
		stState := E_StartupStatus.stDone;
		auxRed := FALSE;		
		auxYellow := FALSE;
		auxGreen := TRUE;

END_CASE;

//   Aplicar comandos calculados às saídas físicas / públicas
Global.K1_out 		:= cmdK01;
Global.K3RedOut 	:= auxRed;
Global.K4YellowOut 	:= auxYellow;
Global.K5GreenOut 	:= auxGreen;

END_FUNCTION_BLOCK

// MainProgram
// DEBUG
// {#define DEBUG_MODE}
PROGRAM MainProgram
(*
    Máquina de estados principal do controlador.
    Fluxo geral:
    START   -> READ    (quando fbStart termina com sucesso)
    READ    -> CONTROL (quando leitura Modbus do medidor conclui OK)
    READ    -> IDLE    (quando leitura falha, mas ainda não estourou RETRIES_READ)
    READ    -> FAIL    (quando leitura falha e estoura RETRIES_READ)
    CONTROL -> WRITE   (sempre, um ciclo de controle por leitura)
    WRITE   -> IDLE    (depois de tentar escrever em todos inversores, se não estourou RETRIES_WRITE)
    WRITE   -> FAIL    (se falhas de escrita estourarem RETRIES_WRITE)
    IDLE    -> READ    (quando completar 1 segundo de ciclo)
    FAIL    -> (aguarda ação do operador)
    STOP    -> (parada controlada, permanece travado)
*)

VAR
    fbStart         		: FB_Startup;        		// executa a inicialização
    fbControle      		: FB_Controle;		 		// módulo de controle
	fbAlarmes				: FB_Alarmes;		 		// converte códigos de erros em mensagens texto
	fbChannel       		: ModbusChannel;
	fbReadMedidor 			: FB_ReadMedidor;
	fbWriteInvCOM1 			: FB_WriteInv;
    fbWriteInvCOM2 			: FB_WriteInv;
	fbEventLog 				: FB_EventLog;    			// Instância única do ring buffer
    fbEventDisplay  		: FB_EventDisplay;			// prepara dados para a IHM
	
	// ══════════════════════════════════════════════════════════
    // Máquina de Estados
    // ══════════════════════════════════════════════════════════
	MachineState 			: E_MachineState := E_MachineState.START;
	MachineState_Last 		: E_MachineState := E_MachineState.START;
    FailState     			: E_FailState := E_FailState.FS_INIT;
	
	// ══════════════════════════════════════════════════════════
	// Variáveis manipuladas pela IHM
	// ══════════════════════════════════════════════════════════
 	HMI_bRefresh    : BOOL;     // Botão "Refresh" na IHM (pulso)
    HMI_nPage       : UINT;     // Página atual (0 = mais recente)
	
    // ══════════════════════════════════════════════════════════
    // STOP: Trip e Reset Manual
    // ══════════════════════════════════════════════════════════
    StopLatch         : BOOL := FALSE;
    StopResetCmd      : BOOL := FALSE;
    StopEntryTime     : UDINT := 0;
    K2_CheckDone      : BOOL := FALSE;
    sMessage_K2       : STRING(100) := '';
    bResetConditionsOK: BOOL := FALSE;
    sResetDenialReason: STRING(255) := '';
    rTrigReset        : R_TRIG;
    tonResetWindow    : TON;
    
    // ══════════════════════════════════════════════════════════
    // Timers Normativos (DIS-NOR-033)
    // ══════════════════════════════════════════════════════════
    ton15s  : TON;   // Hard limit > 15s → STOP
    ton30s  : TON;   // Exportação > LPI por > 30s → STOP
    ton2s   : TON;   // Confirmação K2 aberto

    // ══════════════════════════════════════════════════════════
    // Health Monitoring
    // ══════════════════════════════════════════════════════════
    MedidorOK         : BOOL := FALSE;
    ComOK             : BOOL := FALSE;
    ComOK_COM1        : BOOL := TRUE;
    ComOK_COM2        : BOOL := TRUE;
    InvOnlineCount    : UINT := 0;
    ScanOverrunCount  : UINT := 0;
	FaultLatch        : BOOL := FALSE;
	
    // ══════════════════════════════════════════════════════════
    // Limites Calculados
    // ══════════════════════════════════════════════════════════
    LPI_per_phase_kW  : REAL := 0.0;
    HardLimit_mag     : REAL := 0.0;
    LPI_mag			  : REAL;
	Export_mag		  : REAL;
    // ══════════════════════════════════════════════════════════
    // Validação Cruzada
    // ══════════════════════════════════════════════════════════
    Pt_Last           : REAL := 0.0;
    P_inv_sum         : REAL := 0.0;
    
    // ══════════════════════════════════════════════════════════
    // Escrita em Inversores (Sequencial)
    // ══════════════════════════════════════════════════════════
    InvIndexCOM1      : UINT := 1;
    InvIndexCOM2      : UINT := 1;
    ErrorCountCOM1    : UINT := 0;
    ErrorCountCOM2    : UINT := 0;
    DoneCOM1          : BOOL := FALSE;
    DoneCOM2          : BOOL := FALSE;
    LastErrorIdxCOM1  : UINT := 0;
    LastErrorIdxCOM2  : UINT := 0;
    WriteErrorCOM1    : BOOL := FALSE;
    WriteErrorCOM2    : BOOL := FALSE;
    
    // ══════════════════════════════════════════════════════════
    // Temporização e Watchdog
    // ══════════════════════════════════════════════════════════
    tCycleStart       : UDINT := 0;
    tCycleEnd         : UDINT;
    tCycle            : UDINT;
    tElapsed          : UDINT;
    bFirstScanRead    : BOOL := TRUE;
    MaxCycleTime      : UDINT := 0;
    CycleTimeOverrunCount : UDINT := 0;
    
    // ══════════════════════════════════════════════════════════
    // Debug/Monitor
    // ══════════════════════════════════════════════════════════
    valor             : UN_Convert_Word_To_Real;
    auxvalor          : REAL := 0;
    stStart, stEnd, stCiclo : SYSTIME;
    tStartCom, tCom, tEndCom: SYSTIME;
    tMax              : SYSTIME := 0;
    Gatilho           : BOOL := TRUE;
    rTrigOn           : R_TRIG;
    fTrigOff          : F_TRIG;
    Primeiravez       : BOOL := TRUE;
    stCicloMax        : SYSTIME := 0;
    i                 : UINT;
    
    // ══════════════════════════════════════════════════════════
    // FAIL_SAFE (STOP Timeout)
    // ══════════════════════════════════════════════════════════
    tonStopWrite      : TON;
    tStopWrite        : TIME := T#2S;


	tonFailSafeRecovery		: TON;   // tempo para recuperação ao normal
	tonMedidorTimeout		: TON;   // tempo que aguarda medidor sem leitura
    
END_VAR

// Chama o FB de display todo ciclo (ele só recalcula quando HMI_bRefresh der pulso)
fbEventDisplay(
    pEventLog   := fbEventLog,     // referência ao ring buffer
    bRefresh    := HMI_bRefresh,   // pulso da IHM
    nPageOffset := HMI_nPage       // página selecionada
);


// ════════════════════════════════════════════════════════════════
// MÁQUINA DE ESTADOS PRINCIPAL
// ════════════════════════════════════════════════════════════════
CASE MachineState OF
	
// ────────────────────────────────────────────────────────────────
// START: Inicialização (fbStart + K1/K2)
E_MachineState.START:
    fbStart();  // Chamada do bloco de inicialização
	
	CASE fbStart.stState OF
  		E_StartupStatus.stSeriais,
		E_StartupStatus.stInit,
        E_StartupStatus.stWait_K1,
        E_StartupStatus.stWait_K2:
        	// Permanece em START
        E_StartupStatus.stDone:
			// Inicialização única (executada 1x após power-on)
			FailState := E_FailState.FS_INIT;
			FaultCode := 0;
			FaultLatch := FALSE;
			StopLatch := FALSE;
			ton15s(IN := FALSE);
			ton30s(IN := FALSE);
			ton2s(IN := FALSE);
            (* Inicialização concluída – segue para leitura *)		
            MachineState := E_MachineState.READ;

{#ifdef DEBUG_MODE}			
MachineState := E_MachineState.CONTROL;
auxvalor:=0;
{#endif}
	END_CASE;

// ────────────────────────────────────────────────────────────────
// READ: Leitura do Medidor
E_MachineState.READ:

    // Marca início do ciclo apenas uma vez ao entrar em READ
    IF bFirstScanRead THEN
        tCycleStart := SysTimeCore.SysTimeGetMs();
        bFirstScanRead := FALSE;
    END_IF;	
  	fbReadMedidor(Execute := TRUE);
	// avalia estado do Medidor a cada ciclo
	MedidorOK:=(fbReadMedidor.result = E_ModbusResult.DONE) AND fbReadMedidor.bDadosOK;
    IF fbReadMedidor.result = E_ModbusResult.DONE THEN
		IF MedidorOK THEN
            MachineState := E_MachineState.CONTROL;
        ELSE
            // ❌ Dados inválidos
            IF fbReadMedidor.bPoucosErros THEN
				// Erro isolado → continua com último valor válido
                MachineState := E_MachineState.CONTROL;
                Global.sMessage := 'MEDIÇÃO: Usando último válido';
			ELSE
                // Muitos erros → degradado
                MachineState := E_MachineState.FAIL;
                FaultCode := 16#C1;
                Global.sMessage := 'MEDIÇÃO: Falha persistente';
            END_IF
        END_IF
		
    ELSIF fbReadMedidor.result = E_ModbusResult.ERRO OR fbReadMedidor.result = E_ModbusResult.TIMEOUT THEN
		MachineState := E_MachineState.FAIL; 
        FaultCode := 16#C2;  
    END_IF

// ────────────────────────────────────────────────────────────────
// CONTROL: Cálculo de Setpoints
E_MachineState.CONTROL:
// Calcula setpoints (PI + droop)

IF Global.InstalledPower <= 0.0 THEN
	Global.sMessage := 'ERRO CRITICO: Potencia instalada = 0';
    Global.K8ErroOut := TRUE;
	MachineState := E_MachineState.STOP;
ELSE
	fbControle();  
END_IF

    // Inicialização da Escrita
    IF GVL_Persis.NInversoresCOM01 > 0 THEN
        InvIndexCOM1 := 1;
        DoneCOM1 := FALSE;
    ELSE
        DoneCOM1 := TRUE;
		// SINALIZA ERRO
    END_IF;

    IF GVL_Persis.NInversoresCOM02 > 0 THEN
        InvIndexCOM2 := 1;
        DoneCOM2 := FALSE;
    ELSE
        DoneCOM2 := TRUE;
    END_IF;

    MachineState := E_MachineState.WRITE;
{#ifdef DEBUG_MODE}	
MachineState := E_MachineState.CONTROL;
{#endif}

// ────────────────────────────────────────────────────────────────
// WRITE: Envia Comandos aos Inversores
E_MachineState.WRITE:
// Envia comandos aos inversores

{#ifdef DEBUG_MODE}	
	IF bFirstScanRead THEN
		tCycleStart := SysTimeCore.SysTimeGetMs();
		bFirstScanRead := FALSE;
	END_IF
{#endif}

	DoneCOM1 := (InvIndexCOM1 > GVL_Persis.NInversoresCOM01);
	DoneCOM2 := (InvIndexCOM2 > GVL_Persis.NInversoresCOM02);

    // COM1 (inversores 1..15)
    IF InvIndexCOM1 <= GVL_Persis.NInversoresCOM01 THEN
        IF GVL_Persis.InvActivePower[InvIndexCOM1] > 0.0 THEN
	{#ifdef DEBUG_MODE}
	// medição do tempo de execução
	rTrigOn(CLK := Global.pInversores100[1]^.xBusy);
	fTrigOff(CLK := Global.pInversores100[15]^.xBusy);
	(* Borda de subida → início *)
	IF rTrigOn.Q AND (InvIndexCOM1=1)   THEN
		SysTimeCore.SysTimeGetUs(tStartCom);
		Gatilho := TRUE;  // libera nova medição
	END_IF
	(* Borda de descida → fim *)
	IF fTrigOff.Q AND Gatilho THEN
		SysTimeCore.SysTimeGetUs(tEndCom);
		tCom := tEndCom - tStartCom; 
		IF tCom>tMax THEN
			tMax:=tCom;
		END_IF
		Gatilho := FALSE;
	END_IF
	{#endif}
            fbWriteInvCOM1(
                Execute := TRUE,
                InvIndex := InvIndexCOM1,
                trigInv := Global.trigInvCOM100[InvIndexCOM1],
                pSlave  := Global.pInversores100[InvIndexCOM1]^
            );

            IF (fbWriteInvCOM1.result = E_ModbusResult.DONE) THEN
                InvIndexCOM1 := InvIndexCOM1 + 1;
            ELSIF (fbWriteInvCOM1.result = E_ModbusResult.ERRO) OR
                  (fbWriteInvCOM1.result = E_ModbusResult.TIMEOUT) THEN
                // registra erro e continua
                ErrorCountCOM1 := ErrorCountCOM1 + 1;
                LastErrorIdxCOM1 := InvIndexCOM1;
                InvIndexCOM1 := InvIndexCOM1 + 1;
            END_IF
        ELSE
            // pular inversor inativo
            InvIndexCOM1 := InvIndexCOM1 + 1;
        END_IF
    ELSE
        DoneCOM1 := TRUE;
    END_IF

    // COM2 (inversores 16..30)
    IF InvIndexCOM2 <= GVL_Persis.NInversoresCOM02 THEN
        IF GVL_Persis.InvActivePower[InvIndexCOM2 + 15] > 0.0 THEN
            fbWriteInvCOM2(
                Execute := TRUE,
                InvIndex := InvIndexCOM2,
                trigInv := Global.trigInvCOM200[InvIndexCOM2],
                pSlave  := Global.pInversores200[InvIndexCOM2]^
            );

            IF (fbWriteInvCOM2.result = E_ModbusResult.DONE) THEN
                InvIndexCOM2 := InvIndexCOM2 + 1;
            ELSIF (fbWriteInvCOM2.result = E_ModbusResult.ERRO) OR
                  (fbWriteInvCOM2.result = E_ModbusResult.TIMEOUT) THEN
                // registra erro e continua
                ErrorCountCOM2 := ErrorCountCOM2 + 1;
                LastErrorIdxCOM2 := InvIndexCOM2;
                InvIndexCOM2 := InvIndexCOM2 + 1;
            END_IF
        ELSE
            // pular inversor inativo
            InvIndexCOM2 := InvIndexCOM2 + 1;
        END_IF
    ELSE
        DoneCOM2 := TRUE;
    END_IF

    // Fim da escrita
    IF DoneCOM1 AND DoneCOM2 THEN
        InvIndexCOM1 := 1;
        InvIndexCOM2 := 1;

        // ── Avaliar falhas por canal (>50% = falha do canal) ──
        IF GVL_Persis.NInversoresCOM01 > 0 THEN
            ComOK_COM1 := (ErrorCountCOM1 <= (GVL_Persis.NInversoresCOM01 / 2));
        ELSE
            ComOK_COM1 := TRUE;  // canal não utilizado = OK
        END_IF

        IF GVL_Persis.NInversoresCOM02 > 0 THEN
            ComOK_COM2 := (ErrorCountCOM2 <= (GVL_Persis.NInversoresCOM02 / 2));
        ELSE
            ComOK_COM2 := TRUE;  // canal não utilizado = OK
        END_IF

        // Qualquer canal ativo com falha → FAIL
        IF NOT ComOK_COM1 OR NOT ComOK_COM2 THEN
            FaultCode := 16#C2;
            MachineState := E_MachineState.FAIL;
        ELSE
            MachineState := E_MachineState.IDLE;
        END_IF
		// avalia o estado da comunicação com inversores
		ComOK:= (ComOK_COM1 AND ComOK_COM2);
        // Reset contadores para próximo ciclo
        ErrorCountCOM1 := 0;
        ErrorCountCOM2 := 0;
    END_IF

// ────────────────────────────────────────────────────────────────
// IDLE: Aguarda Completar Ciclo (1s)			
E_MachineState.IDLE:
//  Aguarda completar período de ciclo (1 segundo) depois de
	IF tCycleStart <> 0 THEN
    	tElapsed := SysTimeCore.SysTimeGetMs() - tCycleStart; 					// Calcula tempo desde início do ciclo
	END_IF;
	IF tElapsed >= GLOBAL.CYCLE_TIME_MS THEN
		MachineState := E_MachineState.READ;
		bFirstScanRead := TRUE;
       	// Atualiza estatísticas
       	IF tElapsed > MaxCycleTime THEN
           MaxCycleTime := tElapsed;
       	END_IF;  

	IF tElapsed > Global.CYCLE_TIME_TOLERANCE THEN
		ScanOverrunCount := ScanOverrunCount + 1;
		IF ScanOverrunCount >= 3 THEN
			FaultCode := 16#F1;  						// Watchdog scan
			MachineState := E_MachineState.FAIL;
			Global.sMessage := 'FAIL: Watchdog de ciclo';
			ScanOverrunCount := 0;
		END_IF
	ELSE
		ScanOverrunCount := 0;
	END_IF
{#ifdef DEBUG_MODE}
		MachineState := E_MachineState.CONTROL;
{#endif}
	END_IF;

// ────────────────────────────────────────────────────────────────
E_MachineState.FAIL:
// ESTADO FAIL — Redução forçada (norma DIS-NOR-033)
// ton15s: P > LPI + 10% Pnom por >15s → STOP
// ton30s: P > LPI por >30s → STOP

    // ══════════════════════════════════════════════════════════
    // TIMERS NORMATIVOS (monitorados TODO CICLO)
    // Cálculo do hard limit
	LPI_mag := ABS(Global.MaxExportLimit);
	Export_mag := MAX(0, -Global.Pt);
    HardLimit_mag := LPI_mag + (Global.InstalledPower * 0.1);
	
    // Mantém leitura do medidor (diagnóstico)
    fbReadMedidor(Execute := TRUE);
	
	// ✅ CORREÇÃO: Atualiza MedidorOK dentro de FAIL
    MedidorOK := (fbReadMedidor.result = E_ModbusResult.DONE) AND fbReadMedidor.bDadosOK;	
	
    // ── TIMER 15s: hard limit (P > LPI + 10% Pnom) ──
    ton15s(IN := (Export_mag > HardLimit_mag), PT := T#15S);

    // ── TIMER 30s: exportação persistente (P > LPI) ──
    ton30s(IN := (Export_mag > LPI_mag), PT := T#30S);
	
    // ── Escalada para STOP ──
    IF ton15s.Q OR ton30s.Q THEN
		IF ton15s.Q THEN
			FaultCode := 16#E1;  // hard limit: P > LPI + 10% Pnom por >15s
		ELSIF ton30s.Q THEN
			FaultCode := 16#E2;  // exportação > LPI por >30s
		END_IF
        MachineState := E_MachineState.STOP;
        RETURN;
    END_IF

    // ══════════════════════════════════════════════════════════
    // SUB-ESTADOS SIMPLIFICADOS
    CASE FailState OF

        E_FailState.FS_INIT:
		
			// Sinalização
			Global.K4YellowOut := TRUE;
			Global.K5GreenOut := FALSE;
            // Reinicializa índices de escrita
            InvIndexCOM1 := 1;
            InvIndexCOM2 := 1;
            DoneCOM1 := FALSE;
            DoneCOM2 := FALSE;
			ton15s(IN := FALSE);  
			ton30s(IN := FALSE);
			tonFailSafeRecovery(IN := FALSE);
			tonMedidorTimeout(IN := FALSE); 
            // Zera setpoints
            FOR i := 1 TO Global.NMAXINVERSORES DO
                Global.P_inv_kW[i] := 0.0;
                Global.P_inv_Percent[i] := 0.0;
                Global.Q_inv_kvar[i] := 0.0;
            END_FOR
            FailState := E_FailState.FS_FORCE_ZERO;
			Global.sMessage := 'Entrada em FAIL';

        E_FailState.FS_FORCE_ZERO:
            // Escreve zero em todos os inversores (mesmo código do WRITE, simplificado)
            DoneCOM1 := (InvIndexCOM1 > GVL_Persis.NInversoresCOM01);
            DoneCOM2 := (InvIndexCOM2 > GVL_Persis.NInversoresCOM02);

            // COM1
            IF NOT DoneCOM1 THEN
                IF GVL_Persis.InvActivePower[InvIndexCOM1] > 0.0 THEN
                    fbWriteInvCOM1(
                        Execute := TRUE,
                        InvIndex := InvIndexCOM1,
                        trigInv := Global.trigInvCOM100[InvIndexCOM1],
                        pSlave  := Global.pInversores100[InvIndexCOM1]^
                    );
                    IF (fbWriteInvCOM1.result = E_ModbusResult.DONE) OR
                       (fbWriteInvCOM1.result = E_ModbusResult.ERRO) OR
                       (fbWriteInvCOM1.result = E_ModbusResult.TIMEOUT) THEN
                        InvIndexCOM1 := InvIndexCOM1 + 1;
                    END_IF
                ELSE
                    InvIndexCOM1 := InvIndexCOM1 + 1;
                END_IF
            END_IF

            // COM2
            IF NOT DoneCOM2 THEN
                IF GVL_Persis.InvActivePower[InvIndexCOM2 + 15] > 0.0 THEN
                    fbWriteInvCOM2(
                        Execute := TRUE,
                        InvIndex := InvIndexCOM2,
                        trigInv := Global.trigInvCOM200[InvIndexCOM2],
                        pSlave  := Global.pInversores200[InvIndexCOM2]^
                    );
                    IF (fbWriteInvCOM2.result = E_ModbusResult.DONE) OR
                       (fbWriteInvCOM2.result = E_ModbusResult.ERRO) OR
                       (fbWriteInvCOM2.result = E_ModbusResult.TIMEOUT) THEN
                        InvIndexCOM2 := InvIndexCOM2 + 1;
                    END_IF
                ELSE
                    InvIndexCOM2 := InvIndexCOM2 + 1;
                END_IF
            END_IF

            // Escrita completa?
            IF DoneCOM1 AND DoneCOM2 THEN
                FailState := E_FailState.FS_VALIDATE;
            END_IF

        E_FailState.FS_VALIDATE:
            // Recuperação: P dentro da zona de controle (≤ LPI + 10% Pnom)
            IF (fbReadMedidor.result = E_ModbusResult.DONE) AND (Global.Pt >= -(Global.MaxExportLimit)) AND MedidorOK AND ComOK THEN
			   
				// ✅ Condições OK: conta tempo de recuperação
				tonFailSafeRecovery(IN := TRUE, PT := T#10S);
                IF tonFailSafeRecovery.Q THEN
                    // Recuperação automática
                    FailState := E_FailState.FS_INIT;
                    MachineState := E_MachineState.READ;
                    ton15s(IN := FALSE);
                    ton30s(IN := FALSE);
					tonMedidorTimeout(IN := FALSE);
            		tonFailSafeRecovery(IN := FALSE);
                    Global.K4YellowOut := FALSE;
                    Global.sMessage := 'Recuperação automática';
                END_IF				
            ELSE
        		// ❌ Condições NÃO OK: reseta recuperação e testa timeout
                tonFailSafeRecovery(IN := FALSE);
				// ❌ TIMEOUT de medidor (30s sem leitura válida)
                tonMedidorTimeout(IN := (fbReadMedidor.result <> E_ModbusResult.DONE), PT := T#30S);

                IF tonMedidorTimeout.Q THEN
					// ❌ STOP: Perda de visibilidade da planta
                    FaultCode := 16#E3;
                    MachineState := E_MachineState.STOP;
                    Global.sMessage := 'Timeout medidor em FAIL';
					tonMedidorTimeout(IN := FALSE);  // Reset timer
        			RETURN;
                END_IF
            END_IF
    END_CASE

// ────────────────────────────────────────────────────────────────
E_MachineState.STOP:
    // ══════════════════════════════════════════════════════════
    // A. ENTRADA EM STOP (primeira execução)
    // ══════════════════════════════════════════════════════════
    IF NOT StopLatch THEN
        StopLatch := TRUE;
        StopEntryTime := SysTimeCore.SysTimeGetMs();
        K2_CheckDone := FALSE;
        sMessage_K2 := '';
		        
        // Trip imediato
        Global.K2_out := TRUE;					// aciona trip do disjuntor
        Global.K1_out := FALSE;					// desliga bobina de minima tensão ou contator se existente
        Global.K3RedOut := TRUE;				// indica disjuntor desligado e houve falha
        Global.K4YellowOut := FALSE;
        Global.K5GreenOut := FALSE;
	    // zera setpoints por segurança
        FOR i := 1 TO Global.NMAXINVERSORES DO
            Global.P_inv_kW[i] := 0.0;
            Global.P_inv_Percent[i] := 0.0;
            Global.Q_inv_kvar[i] := 0.0;
        END_FOR	
	
    END_IF
    
    // ══════════════════════════════════════════════════════════
    // B. VERIFICAÇÃO DE K2 (executa apenas 1 vez)
    // ══==══════════════════════════════════════════════════════
    IF NOT K2_CheckDone THEN
        ton2s(IN := TRUE, PT := T#2S);
        
        IF ton2s.Q THEN
            K2_CheckDone := TRUE;
            ton2s(IN := FALSE);
            
            IF Global.K2_in = TRUE THEN
                Global.sMessage := CONCAT('STOP: ', 'CRITICO: K2 não abriu');
                FaultCode := 16#E2;
                FaultLatch := TRUE;
            ELSE
                Global.sMessage := CONCAT('STOP: ','K2 confirmado aberto');
                Global.K4YellowOut := TRUE;
            END_IF
        END_IF
    END_IF
    
    // ══════════════════════════════════════════════════════════
    // C. PROCESSAMENTO DE RESET MANUAL
    // ══════════════════════════════════════════════════════════
    rTrigReset(CLK := StopResetCmd);
    
	// Borda de subida: avalia condições básicas UMA VEZ
    IF rTrigReset.Q THEN
        // Avalia condições básicas
        bResetConditionsOK := (NOT Global.K2_in) AND (NOT FaultLatch) AND MedidorOK AND ComOK;      
		 IF NOT bResetConditionsOK THEN
			// Reset negado imediatamente
			StopResetCmd := FALSE;
			tonResetWindow(IN := FALSE);
			
			IF Global.K2_in THEN
				sResetDenialReason := 'K2 não está aberto';
			ELSIF FaultLatch THEN
				sResetDenialReason := 'FaultLatch ativo';
			ELSE
				sResetDenialReason := 'Medidor não OK';
			END_IF
			
			Global.sMessage := CONCAT('STOP reset NEGADO: ', sResetDenialReason);
		END_IF
	END_IF       
        
	// Monitoramento CONTÍNUO enquanto StopResetCmd=TRUE e condições OK
	IF StopResetCmd AND bResetConditionsOK THEN
		// Timer acumula enquanto Pt dentro do limite
		IF Global.MaxExportLimit > 0.0 THEN
			tonResetWindow(IN := (Global.Pt >= -(Global.MaxExportLimit)), PT := T#10S);
		ELSE
			tonResetWindow(IN := (Global.Pt > 0.0), PT := T#10S);
		END_IF
		
		IF tonResetWindow.Q THEN
			// ✅ Reset aprovado após 10s
			StopLatch := FALSE;
			StopResetCmd := FALSE;
			bResetConditionsOK := FALSE;
			MachineState := E_MachineState.START;
			FaultCode := 0;
			ton15s(IN := FALSE);
			ton30s(IN := FALSE);
			ton2s(IN := FALSE);
			tonResetWindow(IN := FALSE);
			Global.sMessage := 'STOP reset manual OK';
		ELSE
			Global.sMessage := 'Aguardando Pt estável por 10s...';
		END_IF	
	ELSE
		tonResetWindow(IN := FALSE);
	END_IF

END_CASE

END_PROGRAM

// FB Controle/FB_Controle
(*
   FB_Controle: Bloco Principal de Controle de Exportação (Zero Grid / Limitação).
   
   OBJETIVO:
   Gerenciar a potência ativa e reativa dos inversores para garantir que a exportação 
   de energia no ponto de conexão (PCC) não ultrapasse os limites definidos na agenda.

   ESTRATÉGIA DE CONTROLE (Lógica Inversa):
   - PV (Process Variable) é o valor medido no ponto de conexão
     - Valor Positivo (+) = Importando da rede (Consumo > Geração).
     - Valor Negativo (-) = Exportando para rede (Geração > Consumo).
   - SP (Set Point) é o limite de exportação (ex: -50kW).
   - O PID atua para manter PV >= SP.
     - Se PV > SP (Importando), o PID aumenta a geração.
     - Se PV < SP (Exportando), o PID reduz a geração.
	 Controle de Exportação em kW (Zero = Autoconsumo, Negativo = Exportação, Positivo = Importação).
	Erro: SP - PV.
	Ex: Quero exportar -10kW. Medidor lê +5kW (Importando). Erro = -10 - 5 = -15.
	Para aumentar a geração (reduzir a importação), o PID precisa agir. 
	Atenção: Como o comando do inversor é sempre positivo (0..100% de geração), a lógica interna do PI deve ser Inversa (Erro negativo -> Aumenta Saída) ou ajustamos o sinal do erro na entrada.
	
	No código abaixo, a estratégia usada foi de Normalizar o Erro para "Quanto falta gerar".
	Se o medidor diz +10kW (Importando), precisamos gerar +10kW a mais.
	Se o medidor diz -20kW (Exportando muito) e o limite é -10kW, precisamos gerar 10kW a menos.
	
    Hierarquia de prioridades ou objetivos:
	
    Prioridade 1: MAXIMIZAR P (Potência Ativa)
	Objetivo: Gerar o máximo de potência ativa possível
	Limite: Exportação máxima (agenda + safety margin + limite de fase)
	Flexibilidade: RÍGIDO - nunca exceder
	
	Prioridade 2: PF ≥ 0.92 NO PONTO DE CONEXÃO
	Objetivo: Manter fator de potência ≥ 0.92 (indutivo)
	Método: Compensar Q da carga com Q dos inversores
	Flexibilidade: SOFT - sinaliza se não conseguir, mas NÃO reduz P
	
	Prioridade 3: BALANCEAMENTO DE FASES
	
    
    Ordem de execução:
	0. Leitura do medidor e ajuste dos valores para unidades corretas 
	Lê registradores Modbus, converte e armazena como variáveis Globais
	
	Dentro de FB_Controle
	1. FB_Scheduler - Define limite de exportação baseado em datas, dias de semana e horário
    2. FB_PowertController
		2.1. PI → P_cmd_raw
    	2.2. Safety Margin → P_cmd_with_margin
    	2.3. Limitador de Fase → P_cmd_limited 
    3. FB_FFQ - Feedforward de Q (estimativa inicial)
    4. FB_PIQ - Controlador PI de fator de potência
	5. FB_PAlloc - Aloca P pelos inversores 
    6. FB_QAlloc - Aloca Q pelos inversores 
	7. FB_Diagnostico
	8. STATUS DE PF
*)
FUNCTION_BLOCK FB_Controle
VAR_INPUT
    bReset : BOOL;
END_VAR

VAR_OUTPUT
    bPF_OK : BOOL;
END_VAR

VAR
    // ════════════════════════════════════════════════════════════
    // SUBSISTEMAS (Function Blocks)
    // ════════════════════════════════════════════════════════════
    fbScheduler : FB_Scheduler;
    fbPowerCtrl : FB_PowerController;   // ✅ NOVO: Substitui fbPI + fbSafetyMargin + fbFLimiter
    fbFFQ : FB_FFQ;
    fbPIQ : FB_PIQ;
    fbPAlloc : FB_PAlloc;
    fbQAlloc : FB_QAlloc;
    fbDiagnostico : FB_Diagnostico;
    
    // ════════════════════════════════════════════════════════════
    // VARIÁVEIS DE TRABALHO
    // ════════════════════════════════════════════════════════════
    PF_measured : REAL;
    Q_cmd_kvar : REAL;
    Q_feedforward_kvar : REAL;
    bQ_limit_reached : BOOL := FALSE;
    bP_limit_reached : BOOL := FALSE;
END_VAR

// ════════════════════════════════════════════════════════════════
// 0. VERIFICAÇÕES INICIAIS E INICIALIZAÇÃO
// ════════════════════════════════════════════════════════════════
IF Global.InstalledPower <= 0.0 THEN
    // Sem potência instalada: zera todos os comandos
    bPF_OK := FALSE;
    Q_cmd_kvar := 0.0;
    Q_feedforward_kvar := 0.0;
    RETURN;  // Sai sem executar controle
END_IF

IF Global.InstalledSmax <= 0.0 THEN
    // Sem potência aparente: impossível calcular Q
    bPF_OK := FALSE;
    Q_cmd_kvar := 0.0;
    RETURN;
END_IF
// Fator de potência medido (valor absoluto)
PF_measured := ABS(Global.PFt);

// ════════════════════════════════════════════════════════════════
// 1. FB_SCHEDULER - Define Limite de Exportação
// ════════════════════════════════════════════════════════════════

IF GVL_Persis.OperationMode THEN
	Global.MaxExportLimit:=0;				// TRUE = Zero Grid (exportação zero)
ELSE
	fbScheduler();   						// Global.MaxExportLimit definido a partir das agendas de horarios no Scheduller
END_IF

// ────────────────────────────────────────────────────────────────
// 2. CONTROLADOR DE POTÊNCIA ATIVA (PI + Safety + Limites)
// ────────────────────────────────────────────────────────────────

fbPowerCtrl(
    ExportLimit_kW := Global.MaxExportLimit,
    Feedback_kW := Global.Pt,
    bReset := bReset
);

bP_limit_reached := fbPowerCtrl.bPhase_limited OR fbPowerCtrl.bSaturated;
// ════════════════════════════════════════════════════════════════
// 3. FB_FFQ - Feedforward de Q 
// ════════════════════════════════════════════════════════════════

// Calcula Q necessário para manter PF = 0.92 com a potência comandada
fbFFQ(
    P_active_kW := fbPowerCtrl.P_cmd_kW, 
    PF_target_abs := GVL_Persis.PF_target,
    PF_sign := 1.0                              // Indutivo (positivo)
);

Q_feedforward_kvar := fbFFQ.Q_reactive_kvar;  	

// ════════════════════════════════════════════════════════════════
// 4. FB_PIQ - Controle de Fator de Potência
// ════════════════════════════════════════════════════════════════

// Controlador PI de fator de potência
fbPIQ(
    SP := GVL_Persis.PF_target,         							// Setpoint de PF (0.92)
    PV := PF_measured,              							// PF medido (absoluto)
	Kp:= GVL_Persis.Kp_Q,
	Ki:= GVL_Persis.Ki_Q,
	CycleTime:= Global.ControlCycle,
    P_cmd := fbPowerCtrl.P_cmd_kW,     							// Comando de P (para referência)
    RampUp := GVL_Persis.RampUp_Q,      							// Rampa de subida (kvar/s)
    RampDown := GVL_Persis.RampDown_Q,  							// Rampa de descida (kvar/s)
    DeadbandAbs := GVL_Persis.Deadband_Q, 							// Zona morta de PF
    Reset := bReset,                 							// Reset
	bExternal_Saturated := bQ_limit_reached OR bP_limit_reached // FEEDBACK do ciclo anterior - calculado em fbQAlloc.
);

Q_cmd_kvar := Q_feedforward_kvar + fbPIQ.MV;  // Comando de Q em kvar

// Clamp superior: não pode exceder Q máximo dos inversores
IF Q_cmd_kvar > Global.Q_max_permitido THEN
    Q_cmd_kvar := Global.Q_max_permitido;
END_IF
// Clamp inferior: se PF_sign = indutivo, Q não pode ser negativo
IF Q_cmd_kvar < 0.0 THEN
    Q_cmd_kvar := 0.0;  // Não permite Q negativo (capacitivo) se não desejado
END_IF

// ════════════════════════════════════════════════════════════════
// 5. FB_PAlloc - Aloca P (PRIORIDADE MÁXIMA)
// ══════════���═════════════════════════════════════════════════════

fbPAlloc(
    P_total_cmd_kW := fbPowerCtrl.P_cmd_kW
);

Global.P_allocated_kW := fbPAlloc.P_allocated_kW;

// ════════════════════════════════════════════════════════════════
// 6. FB_QAlloc - Aloca Q 
// ════════════════════════════════════════════════════════════════

fbQAlloc(
    Q_total_cmd_kvar := Q_cmd_kvar
);

Global.Q_allocated_kvar := fbQAlloc.Q_allocated_kvar;

// Armazena flag de saturação para próximo ciclo
bQ_limit_reached := fbQAlloc.bQ_limit_reached;

// ════════════════════════════════════════════════════════════════
// 7. FB_Diagnostico - Gera diagnóstico completo
// ════════════════════════════════════════════════════════════════

fbDiagnostico(
    P_allocated_kW := fbPAlloc.P_allocated_kW,
    Q_commanded_kvar := Q_cmd_kvar,
    Q_allocated_kvar := fbQAlloc.Q_allocated_kvar,
    Q_capacity_kvar := fbQAlloc.Q_capacity_total,
    PF_measured := PF_measured,
    PF_achieved := fbQAlloc.PF_effective,
    bQ_limited := fbQAlloc.bQ_limit_reached
);

// ────────────────────────────────────────────────────────────────
// 8. STATUS DE PF
// ────────────────────────────────────────────────────────────────
IF fbQAlloc.PF_effective >= GVL_Persis.PF_target THEN
    bPF_OK := TRUE;
ELSE
    bPF_OK := FALSE;
END_IF

END_FUNCTION_BLOCK

// FB Controle/FB_Scheduler
(*
    FB_Scheduler
    - Agenda semanal: 24 intervalos por dia, 7 dias.
    - Recebe Hora UTC do sistema e converte internamente para LOCAL (Fuso + DST).
    - Feriados/datas especiais sobrescrevem a agenda.
    - Saída: setpoint % da potência instalada.
*)
FUNCTION_BLOCK FB_Scheduler

VAR
    // ════════════════════════════════════════════════════════════
    // VARIÁVEIS DE TIMESTAMP
    // ════════════════════════════════════════════════════════════
    timestampLocal_UDINT : UDINT;           // ✅ Apenas UDINT (sem DINT)
    offsetSeconds : DINT;                   // Offset em segundos (pode ser negativo)
    offsetSeconds_ABS : UDINT;              // Valor absoluto do offset
    
    // ════════════════════════════════════════════════════════════
    // CONVERSÕES DE DATA/HORA
    // ════════════════════════════════════════════════════════════
    dtNowLocal : DATE_AND_TIME;
    dataNowLocal : DATE;
    todNowLocal : TOD;
    todAsDword : DWORD;
    hora : INT;
    diadasemana : INT;
    
    // ════════════════════════════════════════════════════════════
    // CACHE DE DATAS ESPECIAIS (Otimização)
    // ════════════════════════════════════════════════════════════
    lastCheckedDate : DATE := DATE#1970-01-01;      // Última data verificada
    cachedSpecialDateLimit : REAL := -1.0;          // -1 = inválido
    
    // ════════════════════════════════════════════════════════════
    // AUXILIARES
    // ════════════════════════════════════════════════════════════
    i : UINT;
END_VAR


// ════════════════════════════════════════════════════════════════
// 1. LEITURA DO RELÓGIO DO SISTEMA (UTC)
// ════════════════════════════════════════════════════════════════

Global.timestampUTC := TO_UDINT(SysTimeRtcGet(Global.Result));

IF Global.Result <> eResultCode.OK THEN
    // ❌ ERRO: Relógio não disponível
    Global.MaxExportLimit := 0.0;
    Global.sMessage := 'ERRO CRITICO: Falha ao ler RTC';
    Global.K8ErroOut := TRUE;
    RETURN;
END_IF

// ════════════════════════════════════════════════════════════════
// 2. CÁLCULO DO OFFSET TOTAL (Fuso + Horário de Verão)
// ════════════════════════════════════════════════════════════════

// Offset base (fuso horário em segundos)
offsetSeconds := Global.TIMEZONEOFFSET * 3600;  // Ex: -3 * 3600 = -10800

// Adiciona horário de verão se ativo
IF GVL_Persis.bHorarioVerao THEN
    offsetSeconds := offsetSeconds + 3600;      // +1 hora
END_IF

// ════════════════════════════════════════════════════════════════
// 3. APLICA OFFSET AO TIMESTAMP UTC
// ════════════════════════════════════════════════════════════════

// ✅ MÉTODO SEGURO: Usa valor absoluto e subtrai/soma conforme sinal
offsetSeconds_ABS := DINT_TO_UDINT(ABS(offsetSeconds));

IF offsetSeconds < 0 THEN
    // Fuso NEGATIVO (Américas): subtrai
    timestampLocal_UDINT := Global.timestampUTC - offsetSeconds_ABS;
ELSE
    // Fuso POSITIVO (Europa, Ásia): soma
    timestampLocal_UDINT := Global.timestampUTC + offsetSeconds_ABS;
END_IF

// ════════════════════════════════════════════════════════════════
// 4. CONVERTE TIMESTAMP PARA DATA/HORA LOCAL
// ════════════════════════════════════════════════════════════════

dtNowLocal := UDINT_TO_DT(timestampLocal_UDINT);
dataNowLocal := TO_DATE(dtNowLocal);

// Extrai hora (0..23)
todNowLocal := DT_TO_TOD(dtNowLocal);
todAsDword := TOD_TO_DWORD(todNowLocal);
hora := DWORD_TO_INT(todAsDword / DWORD#3600000);

// Extrai dia da semana (1=Dom .. 7=Sáb)
diadasemana := UDINT_TO_INT(((timestampLocal_UDINT / 86400) + 4) MOD 7) + 1;

// ════════════════════════════���═══════════════════════════════════
// 5. VERIFICA MUDANÇA DE DATA (Para atualizar cache)
// ════════════════════════════════════════════════════════════════

IF dataNowLocal <> lastCheckedDate THEN
    
    lastCheckedDate := dataNowLocal;
    cachedSpecialDateLimit := -1.0;  // Invalida cache
    
    FOR i := 1 TO Global.NDATASESPECIAIS DO
        
        // ✅ OTIMIZAÇÃO: Early exit se encontrar data vazia
        IF GVL_Persis.DatasEspeciais[i] = DATE#1970-01-01 THEN
            EXIT;  // Resto do array está vazio
        END_IF
        
        // Verifica se é data especial
        IF GVL_Persis.DatasEspeciais[i] = dataNowLocal THEN
            cachedSpecialDateLimit := GVL_Persis.SpecialDaySchedule[i];
            EXIT;  // Encontrou, pára a busca
        END_IF
        
    END_FOR
    
END_IF

// ════════════════════════════════════════════════════════════════
// 6. USA CACHE DE DATA ESPECIAL (Se válido)
// ════════════════════════════════════════════════════════════════

IF cachedSpecialDateLimit >= 0.0 THEN
    // Data especial ativa
    Global.MaxExportLimit := cachedSpecialDateLimit;
    Global.sMessage := 'Agenda: Data especial';
    RETURN;
END_IF

// ════════════════════════════════════════════════════════════════
// 7. AGENDA SEMANAL (Hora Local)
// ════════════════════════════════════════════════════════════════

// ✅ VALIDAÇÃO: Verifica se índices estão dentro dos limites
IF (diadasemana >= 1 AND diadasemana <= 7) AND (hora >= 0 AND hora <= 23) THEN
    
    // Acessa agenda semanal
    Global.MaxExportLimit := GVL_Persis.WeekSchedule_kW[diadasemana, hora + 1];
    Global.sMessage := '';  // ✅ Limpa mensagem de erro anterior
    
ELSE
    
    // ❌ ERRO: Índice inválido (não deveria ocorrer)
    Global.MaxExportLimit := 0.0;
    Global.sMessage := 'ERRO: Índice de agenda inválido';
    Global.K8ErroOut := TRUE;
    
END_IF

END_FUNCTION_BLOCK

// FB Controle/FB_FFQ
(*
    FB_FFQ - Feedforward de Potência Reativa 
    Função:
    - Calcula o Q MÍNIMO necessário para atingir PF_target
    - Não calcula Q exato, mas o valor mínimo aceitável
    - Se o sistema fornecer menos Q, o PF ficará maior (melhor)
    - Se fornecer mais Q, o PF ficará menor (pior)
    Fórmula:
    Q_min = P × tan(acos(PF_target)) => Simplificado: Q_min = P × √(1 - PF²) / PF
*)

FUNCTION_BLOCK FB_FFQ
VAR_INPUT
    P_active_kW   : REAL;    // Potência ativa comandada (kW)
    PF_target_abs : REAL;    // PF alvo (0.92)
    PF_sign       : REAL;    // 1.0 = indutivo, -1.0 = capacitivo
END_VAR

VAR_OUTPUT
    Q_reactive_kvar : REAL;   // Potência Reativa Calculada (var) - Q mínimo para atingir PF_target
END_VAR

VAR
    tan_phi : REAL;           // Tangente do ângulo de fase
    Q_target    : REAL;       // Q total necessário no ponto de conexão
END_VAR

// 1. Proteção: se potência ativa é zero ou negativa, não há Q a calcular
IF P_active_kW <= 0.0 THEN
    Q_reactive_kvar := 0.0;
    RETURN;
END_IF

// Proteção: PF_target deve estar entre 0 e 1
IF PF_target_abs <= 0.0 OR PF_target_abs > 1.0 THEN
    Q_reactive_kvar := 0.0;
    RETURN;
END_IF

// 2. Q total necessário no ponto de conexão para PF = 0.92
// Método 1: usando tan(acos(PF))
// phi := ACOS(PF_target_abs);              // Ângulo de fase em radianos
// tan_phi := TAN(phi);                     // Tangente do ângulo
// Q_reactive_var := P_active_W * tan_phi;
// Método 2: Simplificado (mais eficiente, evita ACOS e TAN)
// tan(acos(x)) = sqrt(1 - x²) / x
tan_phi := SQRT(1.0 - (PF_target_abs * PF_target_abs)) / PF_target_abs;
Q_target := P_active_kW * tan_phi;

// atribuição correta
Q_reactive_kvar := Q_target;

// 3. Aplica o sinal (Indutivo = positivo, Capacitivo = negativo)
// Nota: Para controle de exportação, normalmente usamos indutivo (Q positivo)
IF PF_sign < 0.0 THEN
    Q_reactive_kvar := -Q_reactive_kvar;  // Capacitivo
END_IF

// Resultado: Q_reactive_var é o Q MÍNIMO para atingir PF_target
// - Se injetar menos Q: PF > PF_target (melhor)
// - Se injetar mais Q: PF < PF_target (pior)
// - Se injetar exatamente Q: PF = PF_target

END_FUNCTION_BLOCK

// FB Controle/FB_PIQ
(*
    FB_PIQ - Controlador PI para Fator de Potência
    Lógica para PF ≥ 0.92:
    - Se PV (PF medido) ≥ SP (PF target): erro = 0 (objetivo atingido)
    - Se PV < SP: erro = SP - PV (precisa aumentar Q)
    Diferente de um PI normal:
    - Erro ZERO quando PF ≥ target (não tenta melhorar além do necessário)
    - Saída é comando de Q (kvar)
*)

FUNCTION_BLOCK FB_PIQ
VAR_INPUT
    SP : REAL;                      		// Setpoint de PF (0.92)
    PV : REAL;                      		// PF medido (absoluto)
	Kp : REAL;              
    Ki : REAL;              
    CycleTime : REAL;       				
    P_cmd : REAL;                   		// Comando de P (para referência)
    RampUp : REAL;                  		// Rampa de subida (kvar/s)
    RampDown : REAL;                		// Rampa de descida (kvar/s)
    DeadbandAbs : REAL;             		// Zona morta de PF (ex: 0.01)
    Reset : BOOL;                   		// Zera o controlador
    bExternal_Saturated : BOOL := FALSE;  	// NOVO: Saturação externa (de FB_QAlloc)
	OutMax : REAL := 1000.0;    			// Limite superior de MV (kvar)
    OutMin : REAL := 0.0;       			// Limite inferior de MV (kvar)
END_VAR

VAR_OUTPUT
    MV : REAL;                      // Comando de Q (kvar)
    Error : REAL;                   // BOOL → REAL (valor do erro)
    Saturated : BOOL;               // TRUE = saída saturada
END_VAR

VAR
    integral : REAL := 0.0;         // Acumulador integral
    P_term : REAL;                  // Termo proporcional
    I_term : REAL;                  // Termo integral
    MV_raw : REAL;                  // Saída bruta (antes de rampa)
    MV_prev : REAL := 0.0;          // Saída do ciclo anterior
    delta : REAL;                   // Variação desejada
    delta_max : REAL;               // Variação máxima permitida
    erro : REAL;                    // Erro de PF
    sinal_saturacao : INT;      	// para anti-windup direcional
END_VAR

// ════════════════════════════════════════════════════════════════
// 1. RESET
// ════════════════════════════════════════════════════════════════
IF Reset THEN
    integral := 0.0;
    MV := 0.0;
    MV_prev := 0.0;
    Error := 0.0;  
    Saturated := FALSE;
    RETURN;
END_IF

// ════════════════════════════════════════════════════════════════
// 2. CALCULA ERRO COM LÓGICA ESPECIAL (PF ≥ TARGET)
// ════════════════════════════════════════════════════════════════

IF PV >= SP THEN
    erro := 0.0;  // PF medido ≥ PF target: objetivo atingido
ELSE
    erro := SP - PV;  // PF medido < PF target: precisa corrigir
END_IF

Error := erro;  // ✅ Saída do erro

// ════════════════════════════════════════════════════════════════
// 3. ZONA MORTA (DEADBAND)
// ════════════════════════════════════════════════════════════════

IF ABS(erro) < DeadbandAbs THEN
    erro := 0.0;
END_IF

// ════════════════════════════════════════════════════════════════
// 4. CÁLCULO PI
// ════════════════════════════════════════════════════════════════

P_term := Kp * erro;
I_term := integral + (Ki * erro * CycleTime);
MV_raw := P_term + I_term;

// ════════════════════════════════════════════════════════════════
// 5. ✅ SATURAÇÃO COM OutMax/OutMin (ALTERAÇÃO)
// ════════════════════════════════════════════════════════════════
IF MV_raw > OutMax THEN
    MV_raw := OutMax;
    sinal_saturacao := 1;
ELSIF MV_raw < OutMin THEN
    MV_raw := OutMin;
    sinal_saturacao := -1;
ELSE
    sinal_saturacao := 0;
END_IF

// ════════════════════════════════════════════════════════════════
// 6. ANTI-WINDUP (Conditional Integration)
// ════════════════════════════════════════════════════════════════

IF bExternal_Saturated OR (sinal_saturacao <> 0) THEN
    // Saturado: só acumula se erro empurra para FORA da saturação
    IF (sinal_saturacao = 1 AND erro < 0.0) OR
       (sinal_saturacao = -1 AND erro > 0.0) THEN
        integral := I_term;  // Permite desacumular
    END_IF
    // Caso contrário: integral permanece (freeze)
    Saturated := TRUE;
ELSE
    integral := I_term;
    Saturated := FALSE;
END_IF

// ════════════════════════════════════════════════════════════════
// 7. RATE LIMITER (Rampa)
// ════════════════════════════════════════════════════════════════

delta := MV_raw - MV_prev;

IF delta > 0.0 THEN
    delta_max := RampUp * Global.ControlCycle;
    IF delta > delta_max THEN
        MV := MV_prev + delta_max;
    ELSE
        MV := MV_raw;
    END_IF
    
ELSIF delta < 0.0 THEN
    delta_max := RampDown * Global.ControlCycle;
    IF ABS(delta) > delta_max THEN
        MV := MV_prev - delta_max;
    ELSE
        MV := MV_raw;
    END_IF
    
ELSE
    MV := MV_raw;
END_IF

MV_prev := MV;

END_FUNCTION_BLOCK

// FB Controle/FB_QAlloc

(*
    ════════════════════════════════════════════════════════════════
    FB_QAlloc - Alocador de Potência Reativa
    ════════════════════════════════════════════════════════════════
*)

FUNCTION_BLOCK FB_QAlloc
VAR_INPUT
    Q_total_cmd_kvar : REAL;        // Comando de Q total (do FB_PIQ)
END_VAR

VAR_OUTPUT
    bQ_limit_reached : BOOL;        // TRUE = Não conseguiu alocar todo Q
    Q_allocated_kvar : REAL;        // Q efetivamente alocado
    PF_effective : REAL;            // PF efetivo total resultante
    Q_capacity_total : REAL;        // Capacidade total de Q disponível (kvar)
    S_total_used : REAL;            // S total utilizado (kVA)
END_VAR

VAR

	// ✅ Acumuladores totais
    Q_total : REAL;
    P_total : REAL;
    Q_capacity_total_internal : REAL;
    S_total_used_internal : REAL;

	// ✅ Variáveis por inversor
    Q_target_i : REAL;
    Q_actual_i : REAL;
    Q_max_i : REAL;
    S_available_i : REAL;
    P_actual_i : REAL;
	
    // ✅ Auxiliares
    i : UINT;
    proportion : REAL;
    S_total : REAL;
    S_i : REAL;  // ✅ S do inversor i (calculado 1 vez)
END_VAR

// ════════════════════════════════════════════════════════════════
// INICIALIZAÇÃO
// ════════════════════════════════════════════════════════════════

Q_total := 0.0;
P_total := 0.0;
Q_capacity_total_internal := 0.0;
S_total_used_internal := 0.0;
bQ_limit_reached := FALSE;

// ════════════════════════════════════════════════════════════════
// LOOP PRINCIPAL
// ════════════════════════════════════════════════════════════════

FOR i := 1 TO Global.NMAXINVERSORES DO
    
    IF GVL_Persis.InvActivePower[i] > 0.0 THEN
        
        // ────────────────────────────────────────────────────────
        // A. LÊ P JÁ ALOCADO
        // ────────────────────────────────────────────────────────
        P_actual_i := Global.P_inv_kW[i];
        
        // ────────────────────────────────────────────────────────
        // B. CALCULA Q MÁXIMO DISPONÍVEL
        // ────────────────────────────────────────────────────────
        S_available_i := GVL_Persis.InvSmaxPower[i];
        
        IF S_available_i > ABS(P_actual_i) THEN
            Q_max_i := SQRT((S_available_i * S_available_i) - (P_actual_i * P_actual_i));
        ELSE
            Q_max_i := 0.0;
        END_IF
        
        Global.Inv_Q_available[i] := Q_max_i;
        
        // ─────────────────────────────────────────���──────────────
        // C. DISTRIBUI Q PROPORCIONALMENTE
        // ────────────────────────────────────────────────────────
        IF Global.P_allocated_kW > 0.01 THEN
            proportion := Global.P_inv_kW[i] / Global.P_allocated_kW;
        ELSE
            proportion := 0.0;
        END_IF
        
        Q_target_i := Q_total_cmd_kvar * proportion;
        
        // ────────────────────────────────────────────────────────
        // D. LIMITA Q AO DISPONÍVEL
        // ────────────────────────────────────────────────────────
        IF ABS(Q_target_i) > Q_max_i THEN
            
            IF Q_target_i >= 0.0 THEN
                Q_actual_i := Q_max_i;
            ELSE
                Q_actual_i := -Q_max_i;
            END_IF
            
            bQ_limit_reached := TRUE;
            Global.Inv_limited[i] := TRUE;
            
        ELSE
            Q_actual_i := Q_target_i;
            Global.Inv_limited[i] := FALSE;
        END_IF
        
        // ────────────────────────────────────────────────────────
        // E. ARMAZENA Q
        // ────────────────────���───────────────────────────────────
        Global.Q_inv_kvar[i] := Q_actual_i;
        
        // ────────────────────────────────────────────────────────
        // F. CALCULA S UTILIZADO (✅ UMA VEZ)
        // ────────────────────────────────────────────────────────
        S_i := SQRT((P_actual_i * P_actual_i) + (Q_actual_i * Q_actual_i));
        
        S_total_used_internal := S_total_used_internal + S_i;
        
        // Utilização de S (%)
        IF S_available_i > 0.0 THEN
            Global.Inv_S_utilization[i] := (S_i / S_available_i) * 100.0;
        ELSE
            Global.Inv_S_utilization[i] := 0.0;
        END_IF
        
        // ────────────────────────────────────────────────────────
        // G. CALCULA PF INDIVIDUAL
        // ────────────────────────────────────────────────────────
        IF S_i > 0.01 THEN
            Global.PF_inv[i] := P_actual_i / S_i;
        ELSE
            Global.PF_inv[i] := 1.0;
        END_IF
        
        // ────────────────────────────────────────────────────────
        // H. ACUMULADORES
        // ────────────────────────────────────────────────────────
        P_total := P_total + P_actual_i;
        Q_total := Q_total + Q_actual_i;
        Q_capacity_total_internal := Q_capacity_total_internal + Q_max_i;
        
    ELSE
        // Inversor inativo
        Global.Q_inv_kvar[i] := 0.0;
        Global.PF_inv[i] := 1.0;
        Global.Inv_Q_available[i] := 0.0;
        Global.Inv_S_utilization[i] := 0.0;
        Global.Inv_limited[i] := FALSE;
    END_IF
    
END_FOR

// ════════════════════════════════════════════════════════════════
// SAÍDAS
// ════════════════════════════════════════════════════════════════

Q_allocated_kvar := Q_total;
Q_capacity_total := Q_capacity_total_internal;
S_total_used := S_total_used_internal;

// PF efetivo total
IF P_total > 0.01 OR ABS(Q_total) > 0.01 THEN
    S_total := SQRT((P_total * P_total) + (Q_total * Q_total));
    PF_effective := P_total / S_total;
ELSE
    PF_effective := 1.0;
END_IF

END_FUNCTION_BLOCK

